LIN {X 0,Y 359.061,Z 1104.275,A -85,B 0,C 180,E1 17031.739,E2 17031.739} C_VEL
LIN {X 0,Y 356.222,Z 1112.102,A -85,B 0,C 180,E1 17028.323,E2 17028.323} C_VEL
LIN {X 0,Y 354.093,Z 1119.043,A -85,B 0,C 180,E1 17024.556,E2 17024.556} C_VEL
LIN {X 0,Y 352.905,Z 1123.818,A -85,B 0,C 180,E1 17021.108,E2 17021.108} C_VEL
LIN {X 0,Y 352.252,Z 1127.627,A -85,B 0,C 180,E1 17017.339,E2 17017.339} C_VEL
LIN {X 0,Y 352.019,Z 1129.695,A -85,B 0,C 180,E1 17013.746,E2 17013.746} C_VEL
LIN {X 0,Y 351.982,Z 1130.473,A -85,B 0,C 180,E1 17010.488,E2 17010.488} C_VEL
LIN {X 0,Y 352.008,Z 1129.935,A -85,B 0,C 180,E1 17006.743,E2 17006.743} C_VEL
LIN {X 0,Y 352.17,Z 1128.245,A -85,B 0,C 180,E1 17003.479,E2 17003.479} C_VEL
LIN {X 0,Y 352.699,Z 1124.946,A -85,B 0,C 180,E1 16999.712,E2 16999.712} C_VEL
LIN {X 0,Y 353.78,Z 1120.188,A -85,B 0,C 180,E1 16996.099,E2 16996.099} C_VEL
LIN {X 0,Y 355.733,Z 1113.699,A -85,B 0,C 180,E1 16992.328,E2 16992.328} C_VEL
LIN {X 0,Y 358.371,Z 1106.105,A -85,B 0,C 180,E1 16988.904,E2 16988.904} C_VEL
LIN {X 0,Y 362.142,Z 1096.54,A -85,B 0,C 180,E1 16985.36,E2 16985.36} C_VEL
LIN {X 0,Y 366.491,Z 1086.054,A -85,B 0,C 180,E1 16982.19,E2 16982.19} C_VEL
LIN {X 0,Y 372.055,Z 1073.212,A -85,B 0,C 180,E1 16978.936,E2 16978.936} C_VEL
LIN {X 0,Y 377.632,Z 1060.335,A -85,B 0,C 180,E1 16976.218,E2 16976.218} C_VEL
LIN {X 0,Y 384.31,Z 1044.71,A -85,B 0,C 180,E1 16973.43,E2 16973.43} C_VEL
LIN {X 0,Y 387.935,Z 1036.089,A -85,B 0,C 180,E1 16972.084,E2 16972.084} C_VEL
LIN {X 0,Y 389.23,Z 1030.919,A -85,B 0,C 180,E1 16971.25,E2 16971.25} C_VEL
LIN {X 0,Y 389.848,Z 1018.215,A -85,B 0,C 180,E1 16968.956,E2 16968.956} C_VEL
LIN {X 0,Y 391.267,Z 1012.649,A -85,B 0,C 180,E1 16968.193,E2 16968.193} C_VEL
LIN {X 0,Y 397.679,Z 995.626,A -85,B 0,C 180,E1 16966.355,E2 16966.355} C_VEL
LIN {X 0,Y 404.403,Z 976.385,A -85,B 0,C 180,E1 16964.595,E2 16964.595} C_VEL
LIN {X 0,Y 410.42,Z 957.139,A -85,B 0,C 180,E1 16963.142,E2 16963.142} C_VEL
LIN {X 0,Y 416.404,Z 935.648,A -85,B 0,C 180,E1 16961.79,E2 16961.79} C_VEL
LIN {X 0,Y 421.3,Z 914.994,A -85,B 0,C 180,E1 16960.743,E2 16960.743} C_VEL
LIN {X 0,Y 425.894,Z 891.963,A -85,B 0,C 180,E1 16959.811,E2 16959.811} C_VEL
LIN {X 0,Y 429.214,Z 870.775,A -85,B 0,C 180,E1 16959.159,E2 16959.159} C_VEL
LIN {X 0,Y 431.994,Z 846.358,A -85,B 0,C 180,E1 16958.605,E2 16958.605} C_VEL
LIN {X 0,Y 442.006,Z 679.643,A -85,B 0,C 180,E1 16955.914,E2 16955.914} C_VEL
LIN {X 0,Y 446.907,Z 597.821,A -85,B 0,C 180,E1 16954.587,E2 16954.587} C_VEL
LIN {X 0,Y 437.742,Z 580.906,A -85,B 0,C 180,E1 16952.156,E2 16952.156} C_VEL
LIN {X 0,Y 428.866,Z 565.701,A -85,B 0,C 180,E1 16949.545,E2 16949.545} C_VEL
LIN {X 0,Y 420.78,Z 552.841,A -85,B 0,C 180,E1 16946.878,E2 16946.878} C_VEL
LIN {X 0,Y 413.2,Z 541.412,A -85,B 0,C 180,E1 16944.026,E2 16944.026} C_VEL
LIN {X 0,Y 406.985,Z 532.513,A -85,B 0,C 180,E1 16941.322,E2 16941.322} C_VEL
LIN {X 0,Y 401.123,Z 524.227,A -85,B 0,C 180,E1 16938.306,E2 16938.306} C_VEL
LIN {X 0,Y 396.734,Z 518.263,A -85,B 0,C 180,E1 16935.57,E2 16935.57} C_VEL
LIN {X 0,Y 393.297,Z 513.694,A -85,B 0,C 180,E1 16932.928,E2 16932.928} C_VEL
LIN {X 0,Y 389.738,Z 508.601,A -85,B 0,C 180,E1 16929.153,E2 16929.153} C_VEL
LIN {X 0,Y 387.106,Z 505.134,A -85,B 0,C 180,E1 16923.258,E2 16923.258} C_VEL
LIN {X 0,Y 387.254,Z 504.707,A -85,B 0,C 180,E1 16919.852,E2 16919.852} C_VEL
LIN {X 0,Y 388.647,Z 506.124,A -85,B 0,C 180,E1 16916.312,E2 16916.312} C_VEL
LIN {X 0,Y 393.194,Z 510.647,A -85,B 0,C 180,E1 16911.076,E2 16911.076} C_VEL
LIN {X 0,Y 398.383,Z 516.743,A -85,B 0,C 180,E1 16907.24,E2 16907.24} C_VEL
LIN {X 0,Y 403.316,Z 522.752,A -85,B 0,C 180,E1 16904.396,E2 16904.396} C_VEL
LIN {X 0,Y 408.456,Z 529.319,A -85,B 0,C 180,E1 16901.887,E2 16901.887} C_VEL
LIN {X 0,Y 414.502,Z 537.176,A -85,B 0,C 180,E1 16899.342,E2 16899.342} C_VEL
LIN {X 0,Y 421.272,Z 546.488,A -85,B 0,C 180,E1 16896.833,E2 16896.833} C_VEL
LIN {X 0,Y 430.458,Z 559.864,A -85,B 0,C 180,E1 16893.847,E2 16893.847} C_VEL
LIN {X 0,Y 439.172,Z 573.641,A -85,B 0,C 180,E1 16891.326,E2 16891.326} C_VEL
LIN {X 0,Y 448.301,Z 589.215,A -85,B 0,C 180,E1 16888.931,E2 16888.931} C_VEL
LIN {X 0,Y 448.71,Z 590.437,A -85,B 0,C 180,E1 16888.814,E2 16888.814} C_VEL
LIN {X 0,Y 434.047,Z 817.562,A -85,B 0,C 180,E1 16885.027,E2 16885.027} C_VEL
LIN {X 0,Y 431.532,Z 850.715,A -85,B 0,C 180,E1 16884.419,E2 16884.419} C_VEL
LIN {X 0,Y 428.713,Z 872.916,A -85,B 0,C 180,E1 16883.861,E2 16883.861} C_VEL
LIN {X 0,Y 424.851,Z 896.32,A -85,B 0,C 180,E1 16883.093,E2 16883.093} C_VEL
LIN {X 0,Y 420.337,Z 918.145,A -85,B 0,C 180,E1 16882.163,E2 16882.163} C_VEL
LIN {X 0,Y 414.997,Z 940.571,A -85,B 0,C 180,E1 16880.99,E2 16880.99} C_VEL
LIN {X 0,Y 409.021,Z 961.94,A -85,B 0,C 180,E1 16879.607,E2 16879.607} C_VEL
LIN {X 0,Y 402.496,Z 983.175,A -85,B 0,C 180,E1 16877.969,E2 16877.969} C_VEL
LIN {X 0,Y 395.82,Z 1002.626,A -85,B 0,C 180,E1 16876.155,E2 16876.155} C_VEL
LIN {X 0,Y 389.09,Z 1021.112,A -85,B 0,C 180,E1 16874.141,E2 16874.141} C_VEL
LIN {X 0,Y 382.174,Z 1038.777,A -85,B 0,C 180,E1 16871.849,E2 16871.849} C_VEL
LIN {X 0,Y 375.67,Z 1054.927,A -85,B 0,C 180,E1 16869.405,E2 16869.405} C_VEL
LIN {X 0,Y 368.791,Z 1071.506,A -85,B 0,C 180,E1 16866.425,E2 16866.425} C_VEL
LIN {X 0,Y 362.918,Z 1085.776,A -85,B 0,C 180,E1 16863.404,E2 16863.404} C_VEL
LIN {X 0,Y 357.509,Z 1099.067,A -85,B 0,C 180,E1 16860.042,E2 16860.042} C_VEL
LIN {X 0,Y 353.277,Z 1110.136,A -85,B 0,C 180,E1 16856.745,E2 16856.745} C_VEL
LIN {X 0,Y 349.514,Z 1120.844,A -85,B 0,C 180,E1 16852.897,E2 16852.897} C_VEL
LIN {X 0,Y 347.053,Z 1128.999,A -85,B 0,C 180,E1 16849.349,E2 16849.349} C_VEL
LIN {X 0,Y 345.234,Z 1136.464,A -85,B 0,C 180,E1 16845.281,E2 16845.281} C_VEL
LIN {X 0,Y 344.401,Z 1141.286,A -85,B 0,C 180,E1 16841.896,E2 16841.896} C_VEL
LIN {X 0,Y 344.011,Z 1145.264,A -85,B 0,C 180,E1 16838.188,E2 16838.188} C_VEL
LIN {X 0,Y 343.957,Z 1147.712,A -85,B 0,C 180,E1 16834.354,E2 16834.354} C_VEL
LIN {X 0,Y 343.97,Z 1148.635,A -85,B 0,C 180,E1 16831.166,E2 16831.166} C_VEL
LIN {X 0,Y 343.967,Z 1148.513,A -85,B 0,C 180,E1 16828.001,E2 16828.001} C_VEL
LIN {X 0,Y 343.947,Z 1147.058,A -85,B 0,C 180,E1 16824.327,E2 16824.327} C_VEL
LIN {X 0,Y 344.078,Z 1144.249,A -85,B 0,C 180,E1 16820.803,E2 16820.803} C_VEL
LIN {X 0,Y 344.527,Z 1140.404,A -85,B 0,C 180,E1 16817.428,E2 16817.428} C_VEL
LIN {X 0,Y 345.74,Z 1134.166,A -85,B 0,C 180,E1 16813.363,E2 16813.363} C_VEL
LIN {X 0,Y 347.557,Z 1127.132,A -85,B 0,C 180,E1 16809.804,E2 16809.804} C_VEL
LIN {X 0,Y 350.529,Z 1117.791,A -85,B 0,C 180,E1 16805.926,E2 16805.926} C_VEL
LIN {X 0,Y 354.257,Z 1107.381,A -85,B 0,C 180,E1 16802.408,E2 16802.408} C_VEL
LIN {X 0,Y 358.961,Z 1095.438,A -85,B 0,C 180,E1 16798.981,E2 16798.981} C_VEL
LIN {X 0,Y 364.403,Z 1081.972,A -85,B 0,C 180,E1 16795.771,E2 16795.771} C_VEL
LIN {X 0,Y 370.807,Z 1066.608,A -85,B 0,C 180,E1 16792.647,E2 16792.647} C_VEL
LIN {X 0,Y 377.109,Z 1051.19,A -85,B 0,C 180,E1 16790.021,E2 16790.021} C_VEL
LIN {X 0,Y 384.057,Z 1033.978,A -85,B 0,C 180,E1 16787.498,E2 16787.498} C_VEL
LIN {X 0,Y 391.091,Z 1015.367,A -85,B 0,C 180,E1 16785.222,E2 16785.222} C_VEL
LIN {X 0,Y 398.22,Z 995.587,A -85,B 0,C 180,E1 16783.162,E2 16783.162} C_VEL
LIN {X 0,Y 404.74,Z 975.569,A -85,B 0,C 180,E1 16781.428,E2 16781.428} C_VEL
LIN {X 0,Y 411.226,Z 954.07,A -85,B 0,C 180,E1 16779.862,E2 16779.862} C_VEL
LIN {X 0,Y 416.89,Z 932.287,A -85,B 0,C 180,E1 16778.565,E2 16778.565} C_VEL
LIN {X 0,Y 422.194,Z 909.086,A -85,B 0,C 180,E1 16777.432,E2 16777.432} C_VEL
LIN {X 0,Y 426.486,Z 886.058,A -85,B 0,C 180,E1 16776.558,E2 16776.558} C_VEL
LIN {X 0,Y 430.113,Z 861.931,A -85,B 0,C 180,E1 16775.851,E2 16775.851} C_VEL
LIN {X 0,Y 432.499,Z 838.378,A -85,B 0,C 180,E1 16775.35,E2 16775.35} C_VEL
LIN {X 0,Y 447.368,Z 608.588,A -85,B 0,C 180,E1 16771.497,E2 16771.497} C_VEL
LIN {X 0,Y 448.503,Z 589.718,A -85,B 0,C 180,E1 16771.165,E2 16771.165} C_VEL
LIN {X 0,Y 439.981,Z 575.175,A -85,B 0,C 180,E1 16768.951,E2 16768.951} C_VEL
LIN {X 0,Y 431.796,Z 562.051,A -85,B 0,C 180,E1 16766.621,E2 16766.621} C_VEL
LIN {X 0,Y 423.202,Z 549.341,A -85,B 0,C 180,E1 16763.904,E2 16763.904} C_VEL
LIN {X 0,Y 415.885,Z 539.147,A -85,B 0,C 180,E1 16761.287,E2 16761.287} C_VEL
LIN {X 0,Y 409.44,Z 530.6,A -85,B 0,C 180,E1 16758.658,E2 16758.658} C_VEL
LIN {X 0,Y 405.218,Z 525.317,A -85,B 0,C 180,E1 16756.707,E2 16756.707} C_VEL
LIN {X 0,Y 401.668,Z 520.808,A -85,B 0,C 180,E1 16754.857,E2 16754.857} C_VEL
LIN {X 0,Y 397.261,Z 515.456,A -85,B 0,C 180,E1 16752.206,E2 16752.206} C_VEL
LIN {X 0,Y 392.273,Z 509.7,A -85,B 0,C 180,E1 16748.354,E2 16748.354} C_VEL
LIN {X 0,Y 387.81,Z 505.149,A -85,B 0,C 180,E1 16742.66,E2 16742.66} C_VEL
LIN {X 0,Y 386.775,Z 504.223,A -85,B 0,C 180,E1 16739.111,E2 16739.111} C_VEL
LIN {X 0,Y 386.947,Z 505.163,A -85,B 0,C 180,E1 16735.702,E2 16735.702} C_VEL
LIN {X 0,Y 390.01,Z 509.049,A -85,B 0,C 180,E1 16730.035,E2 16730.035} C_VEL
LIN {X 0,Y 394.226,Z 515.041,A -85,B 0,C 180,E1 16725.982,E2 16725.982} C_VEL
LIN {X 0,Y 397.728,Z 519.696,A -85,B 0,C 180,E1 16723.496,E2 16723.496} C_VEL
LIN {X 0,Y 402.885,Z 526.813,A -85,B 0,C 180,E1 16720.5,E2 16720.5} C_VEL
LIN {X 0,Y 408.579,Z 534.863,A -85,B 0,C 180,E1 16717.746,E2 16717.746} C_VEL
LIN {X 0,Y 414.522,Z 543.603,A -85,B 0,C 180,E1 16715.259,E2 16715.259} C_VEL
LIN {X 0,Y 421.57,Z 554.129,A -85,B 0,C 180,E1 16712.681,E2 16712.681} C_VEL
LIN {X 0,Y 429.653,Z 567.202,A -85,B 0,C 180,E1 16710.054,E2 16710.054} C_VEL
LIN {X 0,Y 438.52,Z 582.46,A -85,B 0,C 180,E1 16707.483,E2 16707.483} C_VEL
LIN {X 0,Y 446.862,Z 597.937,A -85,B 0,C 180,E1 16705.287,E2 16705.287} C_VEL
LIN {X 0,Y 432.543,Z 837.338,A -85,B 0,C 180,E1 16701.454,E2 16701.454} C_VEL
LIN {X 0,Y 430.479,Z 859.725,A -85,B 0,C 180,E1 16701.013,E2 16701.013} C_VEL
LIN {X 0,Y 426.9,Z 885.077,A -85,B 0,C 180,E1 16700.318,E2 16700.318} C_VEL
LIN {X 0,Y 423.093,Z 905.925,A -85,B 0,C 180,E1 16699.551,E2 16699.551} C_VEL
LIN {X 0,Y 417.989,Z 928.682,A -85,B 0,C 180,E1 16698.482,E2 16698.482} C_VEL
LIN {X 0,Y 412.773,Z 948.636,A -85,B 0,C 180,E1 16697.324,E2 16697.324} C_VEL
LIN {X 0,Y 406.394,Z 969.781,A -85,B 0,C 180,E1 16695.825,E2 16695.825} C_VEL
LIN {X 0,Y 400.067,Z 988.711,A -85,B 0,C 180,E1 16694.212,E2 16694.212} C_VEL
LIN {X 0,Y 393.096,Z 1007.592,A -85,B 0,C 180,E1 16692.273,E2 16692.273} C_VEL
LIN {X 0,Y 386.548,Z 1024.183,A -85,B 0,C 180,E1 16690.263,E2 16690.263} C_VEL
LIN {X 0,Y 379.552,Z 1040.768,A -85,B 0,C 180,E1 16687.866,E2 16687.866} C_VEL
LIN {X 0,Y 373.139,Z 1055.439,A -85,B 0,C 180,E1 16685.367,E2 16685.367} C_VEL
LIN {X 0,Y 366.755,Z 1069.59,A -85,B 0,C 180,E1 16682.486,E2 16682.486} C_VEL
LIN {X 0,Y 361.236,Z 1081.899,A -85,B 0,C 180,E1 16679.518,E2 16679.518} C_VEL
LIN {X 0,Y 356.1,Z 1093.44,A -85,B 0,C 180,E1 16676.158,E2 16676.158} C_VEL
LIN {X 0,Y 352,Z 1103.261,A -85,B 0,C 180,E1 16672.726,E2 16672.726} C_VEL
LIN {X 0,Y 348.749,Z 1111.638,A -85,B 0,C 180,E1 16669.078,E2 16669.078} C_VEL
LIN {X 0,Y 346.409,Z 1118.767,A -85,B 0,C 180,E1 16665.228,E2 16665.228} C_VEL
LIN {X 0,Y 344.974,Z 1124.033,A -85,B 0,C 180,E1 16661.367,E2 16661.367} C_VEL
LIN {X 0,Y 344.278,Z 1127.839,A -85,B 0,C 180,E1 16657.51,E2 16657.51} C_VEL
LIN {X 0,Y 344.026,Z 1129.906,A -85,B 0,C 180,E1 16653.833,E2 16653.833} C_VEL
LIN {X 0,Y 343.986,Z 1130.683,A -85,B 0,C 180,E1 16650.5,E2 16650.5} C_VEL
LIN {X 0,Y 344.014,Z 1130.145,A -85,B 0,C 180,E1 16646.667,E2 16646.667} C_VEL
LIN {X 0,Y 344.189,Z 1128.456,A -85,B 0,C 180,E1 16643.327,E2 16643.327} C_VEL
LIN {X 0,Y 344.762,Z 1125.16,A -85,B 0,C 180,E1 16639.472,E2 16639.472} C_VEL
LIN {X 0,Y 345.911,Z 1120.403,A -85,B 0,C 180,E1 16635.777,E2 16635.777} C_VEL
LIN {X 0,Y 347.986,Z 1113.918,A -85,B 0,C 180,E1 16631.921,E2 16631.921} C_VEL
LIN {X 0,Y 350.775,Z 1106.327,A -85,B 0,C 180,E1 16628.425,E2 16628.425} C_VEL
LIN {X 0,Y 354.763,Z 1096.7,A -85,B 0,C 180,E1 16624.788,E2 16624.788} C_VEL
LIN {X 0,Y 359.314,Z 1086.226,A -85,B 0,C 180,E1 16621.565,E2 16621.565} C_VEL
LIN {X 0,Y 365.092,Z 1073.454,A -85,B 0,C 180,E1 16618.275,E2 16618.275} C_VEL
LIN {X 0,Y 370.883,Z 1060.583,A -85,B 0,C 180,E1 16615.517,E2 16615.517} C_VEL
LIN {X 0,Y 377.812,Z 1044.976,A -85,B 0,C 180,E1 16612.695,E2 16612.695} C_VEL
LIN {X 0,Y 384.289,Z 1029.794,A -85,B 0,C 180,E1 16610.396,E2 16610.396} C_VEL
LIN {X 0,Y 391.267,Z 1012.649,A -85,B 0,C 180,E1 16608.193,E2 16608.193} C_VEL
LIN {X 0,Y 392.706,Z 1006.997,A -85,B 0,C 180,E1 16607.447,E2 16607.447} C_VEL
LIN {X 0,Y 393.841,Z 992.179,A -85,B 0,C 180,E1 16605.237,E2 16605.237} C_VEL
LIN {X 0,Y 395.183,Z 986.942,A -85,B 0,C 180,E1 16604.67,E2 16604.67} C_VEL
LIN {X 0,Y 401.436,Z 968.72,A -85,B 0,C 180,E1 16603.13,E2 16603.13} C_VEL
LIN {X 0,Y 408.259,Z 946.388,A -85,B 0,C 180,E1 16601.574,E2 16601.574} C_VEL
LIN {X 0,Y 413.677,Z 926.027,A -85,B 0,C 180,E1 16600.414,E2 16600.414} C_VEL
LIN {X 0,Y 418.633,Z 903.902,A -85,B 0,C 180,E1 16599.406,E2 16599.406} C_VEL
LIN {X 0,Y 422.618,Z 882.306,A -85,B 0,C 180,E1 16598.629,E2 16598.629} C_VEL
LIN {X 0,Y 425.943,Z 858.501,A -85,B 0,C 180,E1 16597.999,E2 16597.999} C_VEL
LIN {X 0,Y 428.115,Z 834.877,A -85,B 0,C 180,E1 16597.54,E2 16597.54} C_VEL
LIN {X 0,Y 442.467,Z 601.906,A -85,B 0,C 180,E1 16593.803,E2 16593.803} C_VEL
LIN {X 0,Y 434.281,Z 586.594,A -85,B 0,C 180,E1 16591.549,E2 16591.549} C_VEL
LIN {X 0,Y 426.093,Z 572.293,A -85,B 0,C 180,E1 16589.062,E2 16589.062} C_VEL
LIN {X 0,Y 418.175,Z 559.46,A -85,B 0,C 180,E1 16586.369,E2 16586.369} C_VEL
LIN {X 0,Y 410.619,Z 547.848,A -85,B 0,C 180,E1 16583.424,E2 16583.424} C_VEL
LIN {X 0,Y 405.012,Z 539.706,A -85,B 0,C 180,E1 16580.9,E2 16580.9} C_VEL
LIN {X 0,Y 399.558,Z 531.806,A -85,B 0,C 180,E1 16578.01,E2 16578.01} C_VEL
LIN {X 0,Y 395.256,Z 525.844,A -85,B 0,C 180,E1 16575.254,E2 16575.254} C_VEL
LIN {X 0,Y 391.997,Z 521.416,A -85,B 0,C 180,E1 16572.672,E2 16572.672} C_VEL
LIN {X 0,Y 388.661,Z 516.485,A -85,B 0,C 180,E1 16569.029,E2 16569.029} C_VEL
LIN {X 0,Y 386.113,Z 513.037,A -85,B 0,C 180,E1 16563.117,E2 16563.117} C_VEL
LIN {X 0,Y 386.31,Z 512.683,A -85,B 0,C 180,E1 16559.703,E2 16559.703} C_VEL
LIN {X 0,Y 387.663,Z 514.115,A -85,B 0,C 180,E1 16556.303,E2 16556.303} C_VEL
LIN {X 0,Y 391.966,Z 518.445,A -85,B 0,C 180,E1 16551.27,E2 16551.27} C_VEL
LIN {X 0,Y 396.954,Z 524.439,A -85,B 0,C 180,E1 16547.489,E2 16547.489} C_VEL
LIN {X 0,Y 401.673,Z 530.29,A -85,B 0,C 180,E1 16544.7,E2 16544.7} C_VEL
LIN {X 0,Y 406.721,Z 536.861,A -85,B 0,C 180,E1 16542.177,E2 16542.177} C_VEL
LIN {X 0,Y 412.667,Z 544.776,A -85,B 0,C 180,E1 16539.616,E2 16539.616} C_VEL
LIN {X 0,Y 419.077,Z 553.762,A -85,B 0,C 180,E1 16537.188,E2 16537.188} C_VEL
LIN {X 0,Y 427.821,Z 566.732,A -85,B 0,C 180,E1 16534.27,E2 16534.27} C_VEL
LIN {X 0,Y 436.18,Z 580.196,A -85,B 0,C 180,E1 16531.783,E2 16531.783} C_VEL
LIN {X 0,Y 444.153,Z 594.081,A -85,B 0,C 180,E1 16529.622,E2 16529.622} C_VEL
LIN {X 0,Y 428.924,Z 823.697,A -85,B 0,C 180,E1 16525.783,E2 16525.783} C_VEL
LIN {X 0,Y 426.432,Z 853.288,A -85,B 0,C 180,E1 16525.219,E2 16525.219} C_VEL
LIN {X 0,Y 423.499,Z 875.318,A -85,B 0,C 180,E1 16524.652,E2 16524.652} C_VEL
LIN {X 0,Y 419.11,Z 900.128,A -85,B 0,C 180,E1 16523.802,E2 16523.802} C_VEL
LIN {X 0,Y 414.814,Z 920.165,A -85,B 0,C 180,E1 16522.927,E2 16522.927} C_VEL
LIN {X 0,Y 408.772,Z 944.174,A -85,B 0,C 180,E1 16521.626,E2 16521.626} C_VEL
LIN {X 0,Y 403.199,Z 963.438,A -85,B 0,C 180,E1 16520.355,E2 16520.355} C_VEL
LIN {X 0,Y 396.266,Z 985.057,A -85,B 0,C 180,E1 16518.649,E2 16518.649} C_VEL
LIN {X 0,Y 389.677,Z 1003.651,A -85,B 0,C 180,E1 16516.888,E2 16516.888} C_VEL
LIN {X 0,Y 382.289,Z 1023.139,A -85,B 0,C 180,E1 16514.715,E2 16514.715} C_VEL
LIN {X 0,Y 375.203,Z 1040.555,A -85,B 0,C 180,E1 16512.395,E2 16512.395} C_VEL
LIN {X 0,Y 367.954,Z 1057.843,A -85,B 0,C 180,E1 16509.688,E2 16509.688} C_VEL
LIN {X 0,Y 361.467,Z 1072.824,A -85,B 0,C 180,E1 16506.889,E2 16506.889} C_VEL
LIN {X 0,Y 355.185,Z 1087.473,A -85,B 0,C 180,E1 16503.682,E2 16503.682} C_VEL
LIN {X 0,Y 349.717,Z 1100.347,A -85,B 0,C 180,E1 16500.292,E2 16500.292} C_VEL
LIN {X 0,Y 345.114,Z 1111.95,A -85,B 0,C 180,E1 16496.685,E2 16496.685} C_VEL
LIN {X 0,Y 341.623,Z 1121.453,A -85,B 0,C 180,E1 16493.092,E2 16493.092} C_VEL
LIN {X 0,Y 338.898,Z 1130.216,A -85,B 0,C 180,E1 16489.117,E2 16489.117} C_VEL
LIN {X 0,Y 337.232,Z 1136.774,A -85,B 0,C 180,E1 16485.301,E2 16485.301} C_VEL
LIN {X 0,Y 336.391,Z 1141.5,A -85,B 0,C 180,E1 16481.835,E2 16481.835} C_VEL
LIN {X 0,Y 335.991,Z 1145.436,A -85,B 0,C 180,E1 16477.868,E2 16477.868} C_VEL
LIN {X 0,Y 335.961,Z 1147.581,A -85,B 0,C 180,E1 16474.267,E2 16474.267} C_VEL
LIN {X 0,Y 335.971,Z 1148.449,A -85,B 0,C 180,E1 16471.023,E2 16471.023} C_VEL
LIN {X 0,Y 335.953,Z 1148.23,A -85,B 0,C 180,E1 16467.441,E2 16467.441} C_VEL
LIN {X 0,Y 335.972,Z 1146.373,A -85,B 0,C 180,E1 16463.506,E2 16463.506} C_VEL
LIN {X 0,Y 336.148,Z 1143.536,A -85,B 0,C 180,E1 16460.065,E2 16460.065} C_VEL
LIN {X 0,Y 336.839,Z 1138.854,A -85,B 0,C 180,E1 16456.087,E2 16456.087} C_VEL
LIN {X 0,Y 338.253,Z 1132.467,A -85,B 0,C 180,E1 16452.148,E2 16452.148} C_VEL
LIN {X 0,Y 340.676,Z 1124.324,A -85,B 0,C 180,E1 16448.115,E2 16448.115} C_VEL
LIN {X 0,Y 344.01,Z 1114.727,A -85,B 0,C 180,E1 16444.337,E2 16444.337} C_VEL
LIN {X 0,Y 348.454,Z 1103.461,A -85,B 0,C 180,E1 16440.614,E2 16440.614} C_VEL
LIN {X 0,Y 353.465,Z 1091.288,A -85,B 0,C 180,E1 16437.295,E2 16437.295} C_VEL
LIN {X 0,Y 359.585,Z 1077.194,A -85,B 0,C 180,E1 16434.016,E2 16434.016} C_VEL
LIN {X 0,Y 366.059,Z 1062.027,A -85,B 0,C 180,E1 16431.079,E2 16431.079} C_VEL
LIN {X 0,Y 373.309,Z 1045.042,A -85,B 0,C 180,E1 16428.272,E2 16428.272} C_VEL
LIN {X 0,Y 380.437,Z 1027.457,A -85,B 0,C 180,E1 16425.85,E2 16425.85} C_VEL
LIN {X 0,Y 387.94,Z 1008.17,A -85,B 0,C 180,E1 16423.592,E2 16423.592} C_VEL
LIN {X 0,Y 394.682,Z 989.272,A -85,B 0,C 180,E1 16421.747,E2 16421.747} C_VEL
LIN {X 0,Y 401.548,Z 968.592,A -85,B 0,C 180,E1 16420.03,E2 16420.03} C_VEL
LIN {X 0,Y 407.613,Z 947.896,A -85,B 0,C 180,E1 16418.62,E2 16418.62} C_VEL
LIN {X 0,Y 413.327,Z 926.077,A -85,B 0,C 180,E1 16417.374,E2 16417.374} C_VEL
LIN {X 0,Y 418.318,Z 903.333,A -85,B 0,C 180,E1 16416.339,E2 16416.339} C_VEL
LIN {X 0,Y 422.661,Z 879.915,A -85,B 0,C 180,E1 16415.494,E2 16415.494} C_VEL
LIN {X 0,Y 425.998,Z 855.787,A -85,B 0,C 180,E1 16414.852,E2 16414.852} C_VEL
LIN {X 0,Y 428.309,Z 831.084,A -85,B 0,C 180,E1 16414.356,E2 16414.356} C_VEL
LIN {X 0,Y 443.62,Z 599.589,A -85,B 0,C 180,E1 16410.482,E2 16410.482} C_VEL
LIN {X 0,Y 443.957,Z 593.754,A -85,B 0,C 180,E1 16410.373,E2 16410.373} C_VEL
LIN {X 0,Y 434.757,Z 577.99,A -85,B 0,C 180,E1 16407.869,E2 16407.869} C_VEL
LIN {X 0,Y 427.152,Z 565.836,A -85,B 0,C 180,E1 16405.587,E2 16405.587} C_VEL
LIN {X 0,Y 418.177,Z 552.483,A -85,B 0,C 180,E1 16402.567,E2 16402.567} C_VEL
LIN {X 0,Y 410.693,Z 542.113,A -85,B 0,C 180,E1 16399.669,E2 16399.669} C_VEL
LIN {X 0,Y 404.089,Z 533.48,A -85,B 0,C 180,E1 16396.681,E2 16396.681} C_VEL
LIN {X 0,Y 400.05,Z 528.361,A -85,B 0,C 180,E1 16394.548,E2 16394.548} C_VEL
LIN {X 0,Y 395.847,Z 523.157,A -85,B 0,C 180,E1 16391.954,E2 16391.954} C_VEL
LIN {X 0,Y 391.136,Z 517.574,A -85,B 0,C 180,E1 16388.231,E2 16388.231} C_VEL
LIN {X 0,Y 386.829,Z 513.107,A -85,B 0,C 180,E1 16382.667,E2 16382.667} C_VEL
LIN {X 0,Y 385.819,Z 512.156,A -85,B 0,C 180,E1 16379.258,E2 16379.258} C_VEL
LIN {X 0,Y 385.941,Z 513.05,A -85,B 0,C 180,E1 16375.84,E2 16375.84} C_VEL
LIN {X 0,Y 388.918,Z 516.959,A -85,B 0,C 180,E1 16370.156,E2 16370.156} C_VEL
LIN {X 0,Y 392.899,Z 522.741,A -85,B 0,C 180,E1 16366.234,E2 16366.234} C_VEL
LIN {X 0,Y 396.322,Z 527.441,A -85,B 0,C 180,E1 16363.737,E2 16363.737} C_VEL
LIN {X 0,Y 401.266,Z 534.375,A -85,B 0,C 180,E1 16360.796,E2 16360.796} C_VEL
LIN {X 0,Y 406.783,Z 542.37,A -85,B 0,C 180,E1 16358.061,E2 16358.061} C_VEL
LIN {X 0,Y 412.381,Z 550.762,A -85,B 0,C 180,E1 16355.657,E2 16355.657} C_VEL
LIN {X 0,Y 419.21,Z 561.197,A -85,B 0,C 180,E1 16353.09,E2 16353.09} C_VEL
LIN {X 0,Y 426.958,Z 573.958,A -85,B 0,C 180,E1 16350.502,E2 16350.502} C_VEL
LIN {X 0,Y 435.464,Z 588.887,A -85,B 0,C 180,E1 16347.967,E2 16347.967} C_VEL
LIN {X 0,Y 442.306,Z 601.969,A -85,B 0,C 180,E1 16346.092,E2 16346.092} C_VEL
LIN {X 0,Y 427.4,Z 842.164,A -85,B 0,C 180,E1 16342.225,E2 16342.225} C_VEL
LIN {X 0,Y 424.928,Z 865.952,A -85,B 0,C 180,E1 16341.725,E2 16341.725} C_VEL
LIN {X 0,Y 421.435,Z 888.354,A -85,B 0,C 180,E1 16341.066,E2 16341.066} C_VEL
LIN {X 0,Y 417.061,Z 910.907,A -85,B 0,C 180,E1 16340.199,E2 16340.199} C_VEL
LIN {X 0,Y 412.161,Z 931.437,A -85,B 0,C 180,E1 16339.192,E2 16339.192} C_VEL
LIN {X 0,Y 406.281,Z 952.907,A -85,B 0,C 180,E1 16337.904,E2 16337.904} C_VEL
LIN {X 0,Y 400.038,Z 972.572,A -85,B 0,C 180,E1 16336.457,E2 16336.457} C_VEL
LIN {X 0,Y 393.073,Z 992.503,A -85,B 0,C 180,E1 16334.697,E2 16334.697} C_VEL
LIN {X 0,Y 386.229,Z 1010.244,A -85,B 0,C 180,E1 16332.811,E2 16332.811} C_VEL
LIN {X 0,Y 378.645,Z 1028.577,A -85,B 0,C 180,E1 16330.489,E2 16330.489} C_VEL
LIN {X 0,Y 371.95,Z 1043.768,A -85,B 0,C 180,E1 16328.192,E2 16328.192} C_VEL
LIN {X 0,Y 364.345,Z 1060.361,A -85,B 0,C 180,E1 16325.192,E2 16325.192} C_VEL
LIN {X 0,Y 358.314,Z 1073.269,A -85,B 0,C 180,E1 16322.397,E2 16322.397} C_VEL
LIN {X 0,Y 352.239,Z 1086.178,A -85,B 0,C 180,E1 16319.036,E2 16319.036} C_VEL
LIN {X 0,Y 347.248,Z 1097.184,A -85,B 0,C 180,E1 16315.59,E2 16315.59} C_VEL
LIN {X 0,Y 343.112,Z 1106.689,A -85,B 0,C 180,E1 16311.902,E2 16311.902} C_VEL
LIN {X 0,Y 340.078,Z 1114.592,A -85,B 0,C 180,E1 16308.159,E2 16308.159} C_VEL
LIN {X 0,Y 337.944,Z 1120.95,A -85,B 0,C 180,E1 16304.216,E2 16304.216} C_VEL
LIN {X 0,Y 336.725,Z 1125.788,A -85,B 0,C 180,E1 16300.263,E2 16300.263} C_VEL
LIN {X 0,Y 336.181,Z 1128.812,A -85,B 0,C 180,E1 16296.49,E2 16296.49} C_VEL
LIN {X 0,Y 336.005,Z 1130.574,A -85,B 0,C 180,E1 16292.729,E2 16292.729} C_VEL
LIN {X 0,Y 335.987,Z 1130.841,A -85,B 0,C 180,E1 16288.977,E2 16288.977} C_VEL
LIN {X 0,Y 336.043,Z 1130.029,A -85,B 0,C 180,E1 16285.734,E2 16285.734} C_VEL
LIN {X 0,Y 336.361,Z 1127.731,A -85,B 0,C 180,E1 16281.797,E2 16281.797} C_VEL
LIN {X 0,Y 337.13,Z 1123.979,A -85,B 0,C 180,E1 16278.017,E2 16278.017} C_VEL
LIN {X 0,Y 338.715,Z 1118.601,A -85,B 0,C 180,E1 16274.065,E2 16274.065} C_VEL
LIN {X 0,Y 341.134,Z 1111.739,A -85,B 0,C 180,E1 16270.301,E2 16270.301} C_VEL
LIN {X 0,Y 344.771,Z 1102.878,A -85,B 0,C 180,E1 16266.408,E2 16266.408} C_VEL
LIN {X 0,Y 349.148,Z 1092.979,A -85,B 0,C 180,E1 16262.913,E2 16262.913} C_VEL
LIN {X 0,Y 354.875,Z 1080.664,A -85,B 0,C 180,E1 16259.337,E2 16259.337} C_VEL
LIN {X 0,Y 360.418,Z 1068.892,A -85,B 0,C 180,E1 16256.49,E2 16256.49} C_VEL
LIN {X 0,Y 367.498,Z 1053.723,A -85,B 0,C 180,E1 16253.426,E2 16253.426} C_VEL
LIN {X 0,Y 373.828,Z 1039.776,A -85,B 0,C 180,E1 16251.056,E2 16251.056} C_VEL
LIN {X 0,Y 381.254,Z 1022.611,A -85,B 0,C 180,E1 16248.597,E2 16248.597} C_VEL
LIN {X 0,Y 387.922,Z 1006.245,A -85,B 0,C 180,E1 16246.625,E2 16246.625} C_VEL
LIN {X 0,Y 395.183,Z 986.942,A -85,B 0,C 180,E1 16244.67,E2 16244.67} C_VEL
LIN {X 0,Y 396.663,Z 980.881,A -85,B 0,C 180,E1 16244.017,E2 16244.017} C_VEL
LIN {X 0,Y 398.034,Z 964.709,A -85,B 0,C 180,E1 16242.031,E2 16242.031} C_VEL
LIN {X 0,Y 399.243,Z 959.127,A -85,B 0,C 180,E1 16241.546,E2 16241.546} C_VEL
LIN {X 0,Y 405.336,Z 938.745,A -85,B 0,C 180,E1 16240.228,E2 16240.228} C_VEL
LIN {X 0,Y 410.622,Z 917.961,A -85,B 0,C 180,E1 16239.143,E2 16239.143} C_VEL
LIN {X 0,Y 414.997,Z 897.893,A -85,B 0,C 180,E1 16238.292,E2 16238.292} C_VEL
LIN {X 0,Y 419.115,Z 874.164,A -85,B 0,C 180,E1 16237.516,E2 16237.516} C_VEL
LIN {X 0,Y 421.964,Z 852.291,A -85,B 0,C 180,E1 16236.986,E2 16236.986} C_VEL
LIN {X 0,Y 424.436,Z 819.045,A -85,B 0,C 180,E1 16236.406,E2 16236.406} C_VEL
LIN {X 0,Y 437.983,Z 605.742,A -85,B 0,C 180,E1 16232.97,E2 16232.97} C_VEL
LIN {X 0,Y 430.056,Z 590.772,A -85,B 0,C 180,E1 16230.687,E2 16230.687} C_VEL
LIN {X 0,Y 422.778,Z 577.95,A -85,B 0,C 180,E1 16228.384,E2 16228.384} C_VEL
LIN {X 0,Y 415.17,Z 565.379,A -85,B 0,C 180,E1 16225.691,E2 16225.691} C_VEL
LIN {X 0,Y 407.325,Z 553.137,A -85,B 0,C 180,E1 16222.478,E2 16222.478} C_VEL
LIN {X 0,Y 402.648,Z 546.322,A -85,B 0,C 180,E1 16220.269,E2 16220.269} C_VEL
LIN {X 0,Y 397.857,Z 539.223,A -85,B 0,C 180,E1 16217.628,E2 16217.628} C_VEL
LIN {X 0,Y 393.791,Z 533.425,A -85,B 0,C 180,E1 16214.935,E2 16214.935} C_VEL
LIN {X 0,Y 390.703,Z 529.136,A -85,B 0,C 180,E1 16212.414,E2 16212.414} C_VEL
LIN {X 0,Y 387.472,Z 524.264,A -85,B 0,C 180,E1 16208.752,E2 16208.752} C_VEL
LIN {X 0,Y 385.122,Z 520.94,A -85,B 0,C 180,E1 16202.977,E2 16202.977} C_VEL
LIN {X 0,Y 385.368,Z 520.658,A -85,B 0,C 180,E1 16199.554,E2 16199.554} C_VEL
LIN {X 0,Y 386.763,Z 522.219,A -85,B 0,C 180,E1 16196.146,E2 16196.146} C_VEL
LIN {X 0,Y 390.743,Z 526.245,A -85,B 0,C 180,E1 16191.465,E2 16191.465} C_VEL
LIN {X 0,Y 395.533,Z 532.133,A -85,B 0,C 180,E1 16187.74,E2 16187.74} C_VEL
LIN {X 0,Y 400.165,Z 538.013,A -85,B 0,C 180,E1 16184.938,E2 16184.938} C_VEL
LIN {X 0,Y 404.996,Z 544.403,A -85,B 0,C 180,E1 16182.47,E2 16182.47} C_VEL
LIN {X 0,Y 411.003,Z 552.6,A -85,B 0,C 180,E1 16179.827,E2 16179.827} C_VEL
LIN {X 0,Y 417.334,Z 561.706,A -85,B 0,C 180,E1 16177.385,E2 16177.385} C_VEL
LIN {X 0,Y 425.399,Z 573.92,A -85,B 0,C 180,E1 16174.635,E2 16174.635} C_VEL
LIN {X 0,Y 433.322,Z 586.938,A -85,B 0,C 180,E1 16172.217,E2 16172.217} C_VEL
LIN {X 0,Y 439.646,Z 598.208,A -85,B 0,C 180,E1 16170.438,E2 16170.438} C_VEL
LIN {X 0,Y 423.969,Z 828.427,A -85,B 0,C 180,E1 16166.58,E2 16166.58} C_VEL
LIN {X 0,Y 421.594,Z 854.41,A -85,B 0,C 180,E1 16166.071,E2 16166.071} C_VEL
LIN {X 0,Y 418.438,Z 877.262,A -85,B 0,C 180,E1 16165.476,E2 16165.476} C_VEL
LIN {X 0,Y 414.077,Z 900.9,A -85,B 0,C 180,E1 16164.651,E2 16164.651} C_VEL
LIN {X 0,Y 409.667,Z 920.895,A -85,B 0,C 180,E1 16163.772,E2 16163.772} C_VEL
LIN {X 0,Y 403.471,Z 944.739,A -85,B 0,C 180,E1 16162.47,E2 16162.47} C_VEL
LIN {X 0,Y 397.755,Z 963.938,A -85,B 0,C 180,E1 16161.196,E2 16161.196} C_VEL
LIN {X 0,Y 390.318,Z 986.314,A -85,B 0,C 180,E1 16159.407,E2 16159.407} C_VEL
LIN {X 0,Y 383.852,Z 1003.998,A -85,B 0,C 180,E1 16157.714,E2 16157.714} C_VEL
LIN {X 0,Y 375.999,Z 1023.973,A -85,B 0,C 180,E1 16155.454,E2 16155.454} C_VEL
LIN {X 0,Y 368.968,Z 1040.691,A -85,B 0,C 180,E1 16153.199,E2 16153.199} C_VEL
LIN {X 0,Y 361.502,Z 1057.837,A -85,B 0,C 180,E1 16150.48,E2 16150.48} C_VEL
LIN {X 0,Y 354.675,Z 1072.984,A -85,B 0,C 180,E1 16147.609,E2 16147.609} C_VEL
LIN {X 0,Y 348.002,Z 1087.882,A -85,B 0,C 180,E1 16144.274,E2 16144.274} C_VEL
LIN {X 0,Y 342.468,Z 1100.357,A -85,B 0,C 180,E1 16140.922,E2 16140.922} C_VEL
LIN {X 0,Y 337.528,Z 1112.194,A -85,B 0,C 180,E1 16137.143,E2 16137.143} C_VEL
LIN {X 0,Y 333.886,Z 1121.645,A -85,B 0,C 180,E1 16133.472,E2 16133.472} C_VEL
LIN {X 0,Y 331.033,Z 1130.311,A -85,B 0,C 180,E1 16129.406,E2 16129.406} C_VEL
LIN {X 0,Y 329.288,Z 1136.82,A -85,B 0,C 180,E1 16125.499,E2 16125.499} C_VEL
LIN {X 0,Y 328.379,Z 1141.714,A -85,B 0,C 180,E1 16121.772,E2 16121.772} C_VEL
LIN {X 0,Y 327.983,Z 1145.462,A -85,B 0,C 180,E1 16117.709,E2 16117.709} C_VEL
LIN {X 0,Y 327.959,Z 1147.371,A -85,B 0,C 180,E1 16114.371,E2 16114.371} C_VEL
LIN {X 0,Y 327.973,Z 1148.24,A -85,B 0,C 180,E1 16111.048,E2 16111.048} C_VEL
LIN {X 0,Y 327.954,Z 1148.021,A -85,B 0,C 180,E1 16107.379,E2 16107.379} C_VEL
LIN {X 0,Y 327.974,Z 1146.279,A -85,B 0,C 180,E1 16103.523,E2 16103.523} C_VEL
LIN {X 0,Y 328.154,Z 1143.488,A -85,B 0,C 180,E1 16099.998,E2 16099.998} C_VEL
LIN {X 0,Y 328.877,Z 1138.891,A -85,B 0,C 180,E1 16095.923,E2 16095.923} C_VEL
LIN {X 0,Y 330.381,Z 1132.468,A -85,B 0,C 180,E1 16091.837,E2 16091.837} C_VEL
LIN {X 0,Y 332.761,Z 1124.859,A -85,B 0,C 180,E1 16087.938,E2 16087.938} C_VEL
LIN {X 0,Y 336.194,Z 1115.439,A -85,B 0,C 180,E1 16084.075,E2 16084.075} C_VEL
LIN {X 0,Y 340.3,Z 1105.376,A -85,B 0,C 180,E1 16080.614,E2 16080.614} C_VEL
LIN {X 0,Y 345.934,Z 1092.342,A -85,B 0,C 180,E1 16076.887,E2 16076.887} C_VEL
LIN {X 0,Y 351.522,Z 1079.882,A -85,B 0,C 180,E1 16073.885,E2 16073.885} C_VEL
LIN {X 0,Y 358.885,Z 1063.484,A -85,B 0,C 180,E1 16070.563,E2 16070.563} C_VEL
LIN {X 0,Y 365.479,Z 1048.581,A -85,B 0,C 180,E1 16068.017,E2 16068.017} C_VEL
LIN {X 0,Y 373.625,Z 1029.429,A -85,B 0,C 180,E1 16065.264,E2 16065.264} C_VEL
LIN {X 0,Y 380.557,Z 1012.26,A -85,B 0,C 180,E1 16063.187,E2 16063.187} C_VEL
LIN {X 0,Y 388.475,Z 991.143,A -85,B 0,C 180,E1 16061.049,E2 16061.049} C_VEL
LIN {X 0,Y 394.933,Z 972.331,A -85,B 0,C 180,E1 16059.448,E2 16059.448} C_VEL
LIN {X 0,Y 401.897,Z 949.81,A -85,B 0,C 180,E1 16057.862,E2 16057.862} C_VEL
LIN {X 0,Y 407.235,Z 930.121,A -85,B 0,C 180,E1 16056.711,E2 16056.711} C_VEL
LIN {X 0,Y 412.947,Z 905.644,A -85,B 0,C 180,E1 16055.553,E2 16055.553} C_VEL
LIN {X 0,Y 417.144,Z 883.875,A -85,B 0,C 180,E1 16054.747,E2 16054.747} C_VEL
LIN {X 0,Y 421.033,Z 857.852,A -85,B 0,C 180,E1 16054.022,E2 16054.022} C_VEL
LIN {X 0,Y 423.324,Z 835.091,A -85,B 0,C 180,E1 16053.553,E2 16053.553} C_VEL
LIN {X 0,Y 439.13,Z 603.343,A -85,B 0,C 180,E1 16049.659,E2 16049.659} C_VEL
LIN {X 0,Y 439.444,Z 597.744,A -85,B 0,C 180,E1 16049.55,E2 16049.55} C_VEL
LIN {X 0,Y 430.083,Z 581.622,A -85,B 0,C 180,E1 16046.884,E2 16046.884} C_VEL
LIN {X 0,Y 422.535,Z 569.652,A -85,B 0,C 180,E1 16044.501,E2 16044.501} C_VEL
LIN {X 0,Y 415.393,Z 558.919,A -85,B 0,C 180,E1 16041.981,E2 16041.981} C_VEL
LIN {X 0,Y 408.661,Z 549.362,A -85,B 0,C 180,E1 16039.288,E2 16039.288} C_VEL
LIN {X 0,Y 402.267,Z 540.857,A -85,B 0,C 180,E1 16036.313,E2 16036.313} C_VEL
LIN {X 0,Y 398.443,Z 535.912,A -85,B 0,C 180,E1 16034.237,E2 16034.237} C_VEL
LIN {X 0,Y 394.441,Z 530.857,A -85,B 0,C 180,E1 16031.701,E2 16031.701} C_VEL
LIN {X 0,Y 390,Z 525.448,A -85,B 0,C 180,E1 16028.106,E2 16028.106} C_VEL
LIN {X 0,Y 385.782,Z 520.994,A -85,B 0,C 180,E1 16022.525,E2 16022.525} C_VEL
LIN {X 0,Y 384.825,Z 520.105,A -85,B 0,C 180,E1 16019.107,E2 16019.107} C_VEL
LIN {X 0,Y 384.995,Z 521.108,A -85,B 0,C 180,E1 16015.681,E2 16015.681} C_VEL
LIN {X 0,Y 387.827,Z 524.868,A -85,B 0,C 180,E1 16010.278,E2 16010.278} C_VEL
LIN {X 0,Y 391.664,Z 530.58,A -85,B 0,C 180,E1 16006.416,E2 16006.416} C_VEL
LIN {X 0,Y 394.923,Z 535.181,A -85,B 0,C 180,E1 16003.98,E2 16003.98} C_VEL
LIN {X 0,Y 399.658,Z 541.935,A -85,B 0,C 180,E1 16001.095,E2 16001.095} C_VEL
LIN {X 0,Y 404.926,Z 549.757,A -85,B 0,C 180,E1 15998.412,E2 15998.412} C_VEL
LIN {X 0,Y 410.27,Z 557.935,A -85,B 0,C 180,E1 15996.055,E2 15996.055} C_VEL
LIN {X 0,Y 416.869,Z 568.26,A -85,B 0,C 180,E1 15993.504,E2 15993.504} C_VEL
LIN {X 0,Y 424.224,Z 580.591,A -85,B 0,C 180,E1 15990.98,E2 15990.98} C_VEL
LIN {X 0,Y 432.439,Z 595.311,A -85,B 0,C 180,E1 15988.457,E2 15988.457} C_VEL
LIN {X 0,Y 437.841,Z 605.929,A -85,B 0,C 180,E1 15986.918,E2 15986.918} C_VEL
LIN {X 0,Y 422.623,Z 843.405,A -85,B 0,C 180,E1 15983.08,E2 15983.08} C_VEL
LIN {X 0,Y 419.912,Z 867.81,A -85,B 0,C 180,E1 15982.552,E2 15982.552} C_VEL
LIN {X 0,Y 416.459,Z 889.226,A -85,B 0,C 180,E1 15981.915,E2 15981.915} C_VEL
LIN {X 0,Y 411.727,Z 912.626,A -85,B 0,C 180,E1 15980.999,E2 15980.999} C_VEL
LIN {X 0,Y 406.588,Z 933.462,A -85,B 0,C 180,E1 15979.962,E2 15979.962} C_VEL
LIN {X 0,Y 400.098,Z 955.994,A -85,B 0,C 180,E1 15978.568,E2 15978.568} C_VEL
LIN {X 0,Y 394.003,Z 974.556,A -85,B 0,C 180,E1 15977.174,E2 15977.174} C_VEL
LIN {X 0,Y 386.607,Z 994.811,A -85,B 0,C 180,E1 15975.336,E2 15975.336} C_VEL
LIN {X 0,Y 379.614,Z 1012.357,A -85,B 0,C 180,E1 15973.43,E2 15973.43} C_VEL
LIN {X 0,Y 371.89,Z 1030.237,A -85,B 0,C 180,E1 15971.101,E2 15971.101} C_VEL
LIN {X 0,Y 364.77,Z 1045.859,A -85,B 0,C 180,E1 15968.681,E2 15968.681} C_VEL
LIN {X 0,Y 357.35,Z 1061.367,A -85,B 0,C 180,E1 15965.789,E2 15965.789} C_VEL
LIN {X 0,Y 350.751,Z 1075.019,A -85,B 0,C 180,E1 15962.758,E2 15962.758} C_VEL
LIN {X 0,Y 344.584,Z 1087.523,A -85,B 0,C 180,E1 15959.367,E2 15959.367} C_VEL
LIN {X 0,Y 339.46,Z 1098.356,A -85,B 0,C 180,E1 15955.845,E2 15955.845} C_VEL
LIN {X 0,Y 335.388,Z 1107.306,A -85,B 0,C 180,E1 15952.249,E2 15952.249} C_VEL
LIN {X 0,Y 332.112,Z 1115.402,A -85,B 0,C 180,E1 15948.247,E2 15948.247} C_VEL
LIN {X 0,Y 330.088,Z 1121.166,A -85,B 0,C 180,E1 15944.562,E2 15944.562} C_VEL
LIN {X 0,Y 328.787,Z 1126,A -85,B 0,C 180,E1 15940.514,E2 15940.514} C_VEL
LIN {X 0,Y 328.201,Z 1129.024,A -85,B 0,C 180,E1 15936.648,E2 15936.648} C_VEL
LIN {X 0,Y 328.009,Z 1130.784,A -85,B 0,C 180,E1 15932.796,E2 15932.796} C_VEL
LIN {X 0,Y 327.99,Z 1131.051,A -85,B 0,C 180,E1 15928.952,E2 15928.952} C_VEL
LIN {X 0,Y 328.05,Z 1130.239,A -85,B 0,C 180,E1 15925.63,E2 15925.63} C_VEL
LIN {X 0,Y 328.391,Z 1127.943,A -85,B 0,C 180,E1 15921.596,E2 15921.596} C_VEL
LIN {X 0,Y 329.222,Z 1124.192,A -85,B 0,C 180,E1 15917.725,E2 15917.725} C_VEL
LIN {X 0,Y 330.909,Z 1118.818,A -85,B 0,C 180,E1 15913.679,E2 15913.679} C_VEL
LIN {X 0,Y 333.506,Z 1111.875,A -85,B 0,C 180,E1 15909.787,E2 15909.787} C_VEL
LIN {X 0,Y 337.307,Z 1103.102,A -85,B 0,C 180,E1 15905.853,E2 15905.853} C_VEL
LIN {X 0,Y 341.652,Z 1093.708,A -85,B 0,C 180,E1 15902.457,E2 15902.457} C_VEL
LIN {X 0,Y 347.581,Z 1081.52,A -85,B 0,C 180,E1 15898.814,E2 15898.814} C_VEL
LIN {X 0,Y 353.304,Z 1069.819,A -85,B 0,C 180,E1 15895.919,E2 15895.919} C_VEL
LIN {X 0,Y 360.607,Z 1054.808,A -85,B 0,C 180,E1 15892.809,E2 15892.809} C_VEL
LIN {X 0,Y 367.117,Z 1040.949,A -85,B 0,C 180,E1 15890.407,E2 15890.407} C_VEL
LIN {X 0,Y 375.138,Z 1023.083,A -85,B 0,C 180,E1 15887.803,E2 15887.803} C_VEL
LIN {X 0,Y 381.94,Z 1006.904,A -85,B 0,C 180,E1 15885.833,E2 15885.833} C_VEL
LIN {X 0,Y 389.789,Z 986.658,A -85,B 0,C 180,E1 15883.771,E2 15883.771} C_VEL
LIN {X 0,Y 396.264,Z 968.283,A -85,B 0,C 180,E1 15882.218,E2 15882.218} C_VEL
LIN {X 0,Y 399.243,Z 959.127,A -85,B 0,C 180,E1 15881.546,E2 15881.546} C_VEL
LIN {X 0,Y 400.771,Z 952.562,A -85,B 0,C 180,E1 15880.988,E2 15880.988} C_VEL
LIN {X 0,Y 401.708,Z 936.272,A -85,B 0,C 180,E1 15879.306,E2 15879.306} C_VEL
LIN {X 0,Y 402.832,Z 929.441,A -85,B 0,C 180,E1 15878.813,E2 15878.813} C_VEL
LIN {X 0,Y 408.386,Z 906.653,A -85,B 0,C 180,E1 15877.736,E2 15877.736} C_VEL
LIN {X 0,Y 412.618,Z 885.133,A -85,B 0,C 180,E1 15876.944,E2 15876.944} C_VEL
LIN {X 0,Y 416.465,Z 859.821,A -85,B 0,C 180,E1 15876.254,E2 15876.254} C_VEL
LIN {X 0,Y 418.686,Z 837.544,A -85,B 0,C 180,E1 15875.813,E2 15875.813} C_VEL
LIN {X 0,Y 433.644,Z 609.609,A -85,B 0,C 180,E1 15872.131,E2 15872.131} C_VEL
LIN {X 0,Y 425.627,Z 594.41,A -85,B 0,C 180,E1 15869.715,E2 15869.715} C_VEL
LIN {X 0,Y 417.708,Z 580.384,A -85,B 0,C 180,E1 15867.053,E2 15867.053} C_VEL
LIN {X 0,Y 410.328,Z 568.246,A -85,B 0,C 180,E1 15864.243,E2 15864.243} C_VEL
LIN {X 0,Y 404.258,Z 558.862,A -85,B 0,C 180,E1 15861.587,E2 15861.587} C_VEL
LIN {X 0,Y 400.865,Z 553.695,A -85,B 0,C 180,E1 15859.906,E2 15859.906} C_VEL
LIN {X 0,Y 396.305,Z 546.785,A -85,B 0,C 180,E1 15857.321,E2 15857.321} C_VEL
LIN {X 0,Y 392.338,Z 541.006,A -85,B 0,C 180,E1 15854.614,E2 15854.614} C_VEL
LIN {X 0,Y 389.418,Z 536.854,A -85,B 0,C 180,E1 15852.155,E2 15852.155} C_VEL
LIN {X 0,Y 386.404,Z 532.152,A -85,B 0,C 180,E1 15848.632,E2 15848.632} C_VEL
LIN {X 0,Y 384.133,Z 528.843,A -85,B 0,C 180,E1 15842.835,E2 15842.835} C_VEL
LIN {X 0,Y 384.429,Z 528.633,A -85,B 0,C 180,E1 15839.404,E2 15839.404} C_VEL
LIN {X 0,Y 385.781,Z 530.206,A -85,B 0,C 180,E1 15836.136,E2 15836.136} C_VEL
LIN {X 0,Y 389.597,Z 534.174,A -85,B 0,C 180,E1 15831.588,E2 15831.588} C_VEL
LIN {X 0,Y 394.221,Z 539.984,A -85,B 0,C 180,E1 15827.922,E2 15827.922} C_VEL
LIN {X 0,Y 398.543,Z 545.549,A -85,B 0,C 180,E1 15825.247,E2 15825.247} C_VEL
LIN {X 0,Y 403.564,Z 552.321,A -85,B 0,C 180,E1 15822.629,E2 15822.629} C_VEL
LIN {X 0,Y 409.827,Z 561.071,A -85,B 0,C 180,E1 15819.841,E2 15819.841} C_VEL
LIN {X 0,Y 417.013,Z 571.699,A -85,B 0,C 180,E1 15817.068,E2 15817.068} C_VEL
LIN {X 0,Y 425.706,Z 585.448,A -85,B 0,C 180,E1 15814.133,E2 15814.133} C_VEL
LIN {X 0,Y 435.059,Z 601.728,A -85,B 0,C 180,E1 15811.33,E2 15811.33} C_VEL
LIN {X 0,Y 435.199,Z 602.779,A -85,B 0,C 180,E1 15811.264,E2 15811.264} C_VEL
LIN {X 0,Y 418.997,Z 834.051,A -85,B 0,C 180,E1 15807.378,E2 15807.378} C_VEL
LIN {X 0,Y 416.651,Z 857.154,A -85,B 0,C 180,E1 15806.905,E2 15806.905} C_VEL
LIN {X 0,Y 412.942,Z 881.955,A -85,B 0,C 180,E1 15806.23,E2 15806.23} C_VEL
LIN {X 0,Y 408.597,Z 904.189,A -85,B 0,C 180,E1 15805.421,E2 15805.421} C_VEL
LIN {X 0,Y 403.149,Z 927.459,A -85,B 0,C 180,E1 15804.349,E2 15804.349} C_VEL
LIN {X 0,Y 397.369,Z 948.347,A -85,B 0,C 180,E1 15803.147,E2 15803.147} C_VEL
LIN {X 0,Y 390.393,Z 970.598,A -85,B 0,C 180,E1 15801.605,E2 15801.605} C_VEL
LIN {X 0,Y 383.709,Z 989.563,A -85,B 0,C 180,E1 15800.007,E2 15800.007} C_VEL
LIN {X 0,Y 376.299,Z 1009.066,A -85,B 0,C 180,E1 15798.074,E2 15798.074} C_VEL
LIN {X 0,Y 368.555,Z 1027.623,A -85,B 0,C 180,E1 15795.856,E2 15795.856} C_VEL
LIN {X 0,Y 360.716,Z 1045.607,A -85,B 0,C 180,E1 15793.324,E2 15793.324} C_VEL
LIN {X 0,Y 353.324,Z 1061.629,A -85,B 0,C 180,E1 15790.609,E2 15790.609} C_VEL
LIN {X 0,Y 346.194,Z 1077.023,A -85,B 0,C 180,E1 15787.548,E2 15787.548} C_VEL
LIN {X 0,Y 339.617,Z 1090.889,A -85,B 0,C 180,E1 15784.218,E2 15784.218} C_VEL
LIN {X 0,Y 333.843,Z 1103.624,A -85,B 0,C 180,E1 15780.608,E2 15780.608} C_VEL
LIN {X 0,Y 329.151,Z 1114.326,A -85,B 0,C 180,E1 15776.913,E2 15776.913} C_VEL
LIN {X 0,Y 325.409,Z 1123.924,A -85,B 0,C 180,E1 15772.969,E2 15772.969} C_VEL
LIN {X 0,Y 322.676,Z 1131.974,A -85,B 0,C 180,E1 15768.8,E2 15768.8} C_VEL
LIN {X 0,Y 321.067,Z 1138.185,A -85,B 0,C 180,E1 15764.796,E2 15764.796} C_VEL
LIN {X 0,Y 320.217,Z 1142.961,A -85,B 0,C 180,E1 15760.616,E2 15760.616} C_VEL
LIN {X 0,Y 319.989,Z 1145.845,A -85,B 0,C 180,E1 15757,E2 15757} C_VEL
LIN {X 0,Y 319.955,Z 1147.657,A -85,B 0,C 180,E1 15753.225,E2 15753.225} C_VEL
LIN {X 0,Y 319.971,Z 1148.074,A -85,B 0,C 180,E1 15749.284,E2 15749.284} C_VEL
LIN {X 0,Y 319.963,Z 1147.294,A -85,B 0,C 180,E1 15745.878,E2 15745.878} C_VEL
LIN {X 0,Y 319.98,Z 1145.473,A -85,B 0,C 180,E1 15742.458,E2 15742.458} C_VEL
LIN {X 0,Y 320.34,Z 1142.104,A -85,B 0,C 180,E1 15738.477,E2 15738.477} C_VEL
LIN {X 0,Y 321.345,Z 1136.834,A -85,B 0,C 180,E1 15734.294,E2 15734.294} C_VEL
LIN {X 0,Y 323.069,Z 1130.678,A -85,B 0,C 180,E1 15730.472,E2 15730.472} C_VEL
LIN {X 0,Y 326.157,Z 1121.781,A -85,B 0,C 180,E1 15726.13,E2 15726.13} C_VEL
LIN {X 0,Y 329.753,Z 1112.849,A -85,B 0,C 180,E1 15722.555,E2 15722.555} C_VEL
LIN {X 0,Y 335.1,Z 1100.627,A -85,B 0,C 180,E1 15718.522,E2 15718.522} C_VEL
LIN {X 0,Y 340.532,Z 1088.847,A -85,B 0,C 180,E1 15715.275,E2 15715.275} C_VEL
LIN {X 0,Y 347.768,Z 1073.376,A -85,B 0,C 180,E1 15711.714,E2 15711.714} C_VEL
LIN {X 0,Y 354.525,Z 1058.909,A -85,B 0,C 180,E1 15708.917,E2 15708.917} C_VEL
LIN {X 0,Y 362.581,Z 1041.128,A -85,B 0,C 180,E1 15706.035,E2 15706.035} C_VEL
LIN {X 0,Y 369.752,Z 1024.618,A -85,B 0,C 180,E1 15703.778,E2 15703.778} C_VEL
LIN {X 0,Y 377.824,Z 1004.787,A -85,B 0,C 180,E1 15701.501,E2 15701.501} C_VEL
LIN {X 0,Y 384.623,Z 986.739,A -85,B 0,C 180,E1 15699.756,E2 15699.756} C_VEL
LIN {X 0,Y 392.086,Z 965.028,A -85,B 0,C 180,E1 15698,E2 15698} C_VEL
LIN {X 0,Y 397.935,Z 945.962,A -85,B 0,C 180,E1 15696.721,E2 15696.721} C_VEL
LIN {X 0,Y 403.97,Z 923.746,A -85,B 0,C 180,E1 15695.479,E2 15695.479} C_VEL
LIN {X 0,Y 408.92,Z 902.014,A -85,B 0,C 180,E1 15694.509,E2 15694.509} C_VEL
LIN {X 0,Y 413.461,Z 878.273,A -85,B 0,C 180,E1 15693.67,E2 15693.67} C_VEL
LIN {X 0,Y 416.777,Z 854.903,A -85,B 0,C 180,E1 15693.058,E2 15693.058} C_VEL
LIN {X 0,Y 419.2,Z 829.39,A -85,B 0,C 180,E1 15692.554,E2 15692.554} C_VEL
LIN {X 0,Y 435.087,Z 602.117,A -85,B 0,C 180,E1 15688.738,E2 15688.738} C_VEL
LIN {X 0,Y 427.406,Z 588.495,A -85,B 0,C 180,E1 15686.466,E2 15686.466} C_VEL
LIN {X 0,Y 420.175,Z 576.811,A -85,B 0,C 180,E1 15684.124,E2 15684.124} C_VEL
LIN {X 0,Y 413.165,Z 566.044,A -85,B 0,C 180,E1 15681.583,E2 15681.583} C_VEL
LIN {X 0,Y 406.497,Z 556.411,A -85,B 0,C 180,E1 15678.835,E2 15678.835} C_VEL
LIN {X 0,Y 400.33,Z 548.072,A -85,B 0,C 180,E1 15675.872,E2 15675.872} C_VEL
LIN {X 0,Y 396.97,Z 543.591,A -85,B 0,C 180,E1 15673.993,E2 15673.993} C_VEL
LIN {X 0,Y 393.042,Z 538.556,A -85,B 0,C 180,E1 15671.445,E2 15671.445} C_VEL
LIN {X 0,Y 388.712,Z 533.199,A -85,B 0,C 180,E1 15667.836,E2 15667.836} C_VEL
LIN {X 0,Y 384.739,Z 528.881,A -85,B 0,C 180,E1 15662.383,E2 15662.383} C_VEL
LIN {X 0,Y 383.834,Z 528.053,A -85,B 0,C 180,E1 15658.955,E2 15658.955} C_VEL
LIN {X 0,Y 384.053,Z 529.163,A -85,B 0,C 180,E1 15655.52,E2 15655.52} C_VEL
LIN {X 0,Y 386.739,Z 532.776,A -85,B 0,C 180,E1 15650.4,E2 15650.4} C_VEL
LIN {X 0,Y 390.347,Z 538.278,A -85,B 0,C 180,E1 15646.671,E2 15646.671} C_VEL
LIN {X 0,Y 393.433,Z 542.738,A -85,B 0,C 180,E1 15644.296,E2 15644.296} C_VEL
LIN {X 0,Y 398.184,Z 549.679,A -85,B 0,C 180,E1 15641.327,E2 15641.327} C_VEL
LIN {X 0,Y 403.156,Z 557.258,A -85,B 0,C 180,E1 15638.732,E2 15638.732} C_VEL
LIN {X 0,Y 408.161,Z 565.079,A -85,B 0,C 180,E1 15636.465,E2 15636.465} C_VEL
LIN {X 0,Y 414.553,Z 575.32,A -85,B 0,C 180,E1 15633.923,E2 15633.923} C_VEL
LIN {X 0,Y 421.56,Z 587.298,A -85,B 0,C 180,E1 15631.449,E2 15631.449} C_VEL
LIN {X 0,Y 429.419,Z 601.693,A -85,B 0,C 180,E1 15628.96,E2 15628.96} C_VEL
LIN {X 0,Y 433.473,Z 609.785,A -85,B 0,C 180,E1 15627.763,E2 15627.763} C_VEL
LIN {X 0,Y 417.999,Z 843.958,A -85,B 0,C 180,E1 15623.967,E2 15623.967} C_VEL
LIN {X 0,Y 415.064,Z 869.14,A -85,B 0,C 180,E1 15623.413,E2 15623.413} C_VEL
LIN {X 0,Y 411.546,Z 890.282,A -85,B 0,C 180,E1 15622.778,E2 15622.778} C_VEL
LIN {X 0,Y 406.749,Z 913.197,A -85,B 0,C 180,E1 15621.873,E2 15621.873} C_VEL
LIN {X 0,Y 401.694,Z 933.19,A -85,B 0,C 180,E1 15620.878,E2 15620.878} C_VEL
LIN {X 0,Y 395.124,Z 955.513,A -85,B 0,C 180,E1 15619.503,E2 15619.503} C_VEL
LIN {X 0,Y 388.859,Z 974.13,A -85,B 0,C 180,E1 15618.108,E2 15618.108} C_VEL
LIN {X 0,Y 380.98,Z 995.138,A -85,B 0,C 180,E1 15616.199,E2 15616.199} C_VEL
LIN {X 0,Y 373.784,Z 1012.665,A -85,B 0,C 180,E1 15614.282,E2 15614.282} C_VEL
LIN {X 0,Y 365.821,Z 1030.517,A -85,B 0,C 180,E1 15611.935,E2 15611.935} C_VEL
LIN {X 0,Y 358.468,Z 1046.13,A -85,B 0,C 180,E1 15609.492,E2 15609.492} C_VEL
LIN {X 0,Y 351.158,Z 1060.862,A -85,B 0,C 180,E1 15606.724,E2 15606.724} C_VEL
LIN {X 0,Y 344.648,Z 1073.76,A -85,B 0,C 180,E1 15603.851,E2 15603.851} C_VEL
LIN {X 0,Y 338.063,Z 1086.635,A -85,B 0,C 180,E1 15600.383,E2 15600.383} C_VEL
LIN {X 0,Y 332.594,Z 1097.647,A -85,B 0,C 180,E1 15596.805,E2 15596.805} C_VEL
LIN {X 0,Y 328.031,Z 1107.136,A -85,B 0,C 180,E1 15592.965,E2 15592.965} C_VEL
LIN {X 0,Y 324.521,Z 1115.326,A -85,B 0,C 180,E1 15588.876,E2 15588.876} C_VEL
LIN {X 0,Y 322.243,Z 1121.382,A -85,B 0,C 180,E1 15584.924,E2 15584.924} C_VEL
LIN {X 0,Y 320.855,Z 1126.213,A -85,B 0,C 180,E1 15580.777,E2 15580.777} C_VEL
LIN {X 0,Y 320.218,Z 1129.245,A -85,B 0,C 180,E1 15576.798,E2 15576.798} C_VEL
LIN {X 0,Y 320.013,Z 1130.995,A -85,B 0,C 180,E1 15572.866,E2 15572.866} C_VEL
LIN {X 0,Y 319.993,Z 1131.261,A -85,B 0,C 180,E1 15568.926,E2 15568.926} C_VEL
LIN {X 0,Y 320.058,Z 1130.45,A -85,B 0,C 180,E1 15565.52,E2 15565.52} C_VEL
LIN {X 0,Y 320.423,Z 1128.155,A -85,B 0,C 180,E1 15561.385,E2 15561.385} C_VEL
LIN {X 0,Y 321.321,Z 1124.406,A -85,B 0,C 180,E1 15557.419,E2 15557.419} C_VEL
LIN {X 0,Y 323.117,Z 1119.035,A -85,B 0,C 180,E1 15553.274,E2 15553.274} C_VEL
LIN {X 0,Y 325.832,Z 1112.176,A -85,B 0,C 180,E1 15549.335,E2 15549.335} C_VEL
LIN {X 0,Y 329.875,Z 1103.326,A -85,B 0,C 180,E1 15545.273,E2 15545.273} C_VEL
LIN {X 0,Y 334.43,Z 1093.935,A -85,B 0,C 180,E1 15541.81,E2 15541.81} C_VEL
LIN {X 0,Y 340.621,Z 1081.756,A -85,B 0,C 180,E1 15538.103,E2 15538.103} C_VEL
LIN {X 0,Y 346.94,Z 1069.371,A -85,B 0,C 180,E1 15535.004,E2 15535.004} C_VEL
LIN {X 0,Y 354.558,Z 1054.233,A -85,B 0,C 180,E1 15531.859,E2 15531.859} C_VEL
LIN {X 0,Y 361.332,Z 1040.3,A -85,B 0,C 180,E1 15529.435,E2 15529.435} C_VEL
LIN {X 0,Y 369.656,Z 1022.275,A -85,B 0,C 180,E1 15526.816,E2 15526.816} C_VEL
LIN {X 0,Y 376.885,Z 1005.574,A -85,B 0,C 180,E1 15524.79,E2 15524.79} C_VEL
LIN {X 0,Y 384.532,Z 986.271,A -85,B 0,C 180,E1 15522.838,E2 15522.838} C_VEL
LIN {X 0,Y 391.478,Z 967.061,A -85,B 0,C 180,E1 15521.222,E2 15521.222} C_VEL
LIN {X 0,Y 398.131,Z 946.169,A -85,B 0,C 180,E1 15519.78,E2 15519.78} C_VEL
LIN {X 0,Y 402.832,Z 929.441,A -85,B 0,C 180,E1 15518.813,E2 15518.813} C_VEL
LIN {X 0,Y 404.098,Z 922.514,A -85,B 0,C 180,E1 15518.345,E2 15518.345} C_VEL
LIN {X 0,Y 404.615,Z 905.262,A -85,B 0,C 180,E1 15516.884,E2 15516.884} C_VEL
LIN {X 0,Y 405.533,Z 898.12,A -85,B 0,C 180,E1 15516.481,E2 15516.481} C_VEL
LIN {X 0,Y 409.881,Z 874.28,A -85,B 0,C 180,E1 15515.704,E2 15515.704} C_VEL
LIN {X 0,Y 412.859,Z 852.461,A -85,B 0,C 180,E1 15515.176,E2 15515.176} C_VEL
LIN {X 0,Y 415.467,Z 819.512,A -85,B 0,C 180,E1 15514.598,E2 15514.598} C_VEL
LIN {X 0,Y 429.351,Z 613.526,A -85,B 0,C 180,E1 15511.265,E2 15511.265} C_VEL
LIN {X 0,Y 421.32,Z 598.124,A -85,B 0,C 180,E1 15508.723,E2 15508.723} C_VEL
LIN {X 0,Y 414.29,Z 585.732,A -85,B 0,C 180,E1 15506.249,E2 15506.249} C_VEL
LIN {X 0,Y 408.132,Z 575.285,A -85,B 0,C 180,E1 15503.805,E2 15503.805} C_VEL
LIN {X 0,Y 402.345,Z 566.13,A -85,B 0,C 180,E1 15501.198,E2 15501.198} C_VEL
LIN {X 0,Y 398.331,Z 559.867,A -85,B 0,C 180,E1 15499.122,E2 15499.122} C_VEL
LIN {X 0,Y 394.422,Z 553.93,A -85,B 0,C 180,E1 15496.798,E2 15496.798} C_VEL
LIN {X 0,Y 390.991,Z 548.703,A -85,B 0,C 180,E1 15494.363,E2 15494.363} C_VEL
LIN {X 0,Y 388.14,Z 544.572,A -85,B 0,C 180,E1 15491.893,E2 15491.893} C_VEL
LIN {X 0,Y 385.335,Z 540.036,A -85,B 0,C 180,E1 15488.506,E2 15488.506} C_VEL
LIN {X 0,Y 383.147,Z 536.746,A -85,B 0,C 180,E1 15482.692,E2 15482.692} C_VEL
LIN {X 0,Y 383.454,Z 536.577,A -85,B 0,C 180,E1 15479.402,E2 15479.402} C_VEL
LIN {X 0,Y 384.719,Z 538.082,A -85,B 0,C 180,E1 15476.275,E2 15476.275} C_VEL
LIN {X 0,Y 388.38,Z 541.981,A -85,B 0,C 180,E1 15471.785,E2 15471.785} C_VEL
LIN {X 0,Y 392.814,Z 547.674,A -85,B 0,C 180,E1 15468.176,E2 15468.176} C_VEL
LIN {X 0,Y 397.051,Z 553.267,A -85,B 0,C 180,E1 15465.489,E2 15465.489} C_VEL
LIN {X 0,Y 401.856,Z 559.859,A -85,B 0,C 180,E1 15462.926,E2 15462.926} C_VEL
LIN {X 0,Y 408.571,Z 569.39,A -85,B 0,C 180,E1 15459.889,E2 15459.889} C_VEL
LIN {X 0,Y 416.771,Z 582.034,A -85,B 0,C 180,E1 15456.718,E2 15456.718} C_VEL
LIN {X 0,Y 424.431,Z 594.686,A -85,B 0,C 180,E1 15454.124,E2 15454.124} C_VEL
LIN {X 0,Y 430.922,Z 606.398,A -85,B 0,C 180,E1 15452.123,E2 15452.123} C_VEL
LIN {X 0,Y 414.27,Z 837.139,A -85,B 0,C 180,E1 15448.236,E2 15448.236} C_VEL
LIN {X 0,Y 411.834,Z 859.614,A -85,B 0,C 180,E1 15447.766,E2 15447.766} C_VEL
LIN {X 0,Y 407.778,Z 884.984,A -85,B 0,C 180,E1 15447.049,E2 15447.049} C_VEL
LIN {X 0,Y 403.293,Z 907.039,A -85,B 0,C 180,E1 15446.228,E2 15446.228} C_VEL
LIN {X 0,Y 397.438,Z 930.66,A -85,B 0,C 180,E1 15445.102,E2 15445.102} C_VEL
LIN {X 0,Y 391.625,Z 950.941,A -85,B 0,C 180,E1 15443.909,E2 15443.909} C_VEL
LIN {X 0,Y 384.159,Z 973.592,A -85,B 0,C 180,E1 15442.29,E2 15442.29} C_VEL
LIN {X 0,Y 377.375,Z 992.189,A -85,B 0,C 180,E1 15440.686,E2 15440.686} C_VEL
LIN {X 0,Y 368.863,Z 1013.375,A -85,B 0,C 180,E1 15438.494,E2 15438.494} C_VEL
LIN {X 0,Y 361.4,Z 1030.66,A -85,B 0,C 180,E1 15436.355,E2 15436.355} C_VEL
LIN {X 0,Y 353.025,Z 1048.895,A -85,B 0,C 180,E1 15433.66,E2 15433.66} C_VEL
LIN {X 0,Y 345.806,Z 1064.034,A -85,B 0,C 180,E1 15431.003,E2 15431.003} C_VEL
LIN {X 0,Y 338.194,Z 1079.647,A -85,B 0,C 180,E1 15427.735,E2 15427.735} C_VEL
LIN {X 0,Y 332.155,Z 1091.948,A -85,B 0,C 180,E1 15424.677,E2 15424.677} C_VEL
LIN {X 0,Y 325.694,Z 1105.507,A -85,B 0,C 180,E1 15420.639,E2 15420.639} C_VEL
LIN {X 0,Y 321.172,Z 1115.513,A -85,B 0,C 180,E1 15417.035,E2 15417.035} C_VEL
LIN {X 0,Y 317.079,Z 1125.557,A -85,B 0,C 180,E1 15412.627,E2 15412.627} C_VEL
LIN {X 0,Y 314.706,Z 1132.382,A -85,B 0,C 180,E1 15408.91,E2 15408.91} C_VEL
LIN {X 0,Y 312.985,Z 1138.801,A -85,B 0,C 180,E1 15404.535,E2 15404.535} C_VEL
LIN {X 0,Y 312.204,Z 1143.091,A -85,B 0,C 180,E1 15400.508,E2 15400.508} C_VEL
LIN {X 0,Y 311.98,Z 1145.871,A -85,B 0,C 180,E1 15396.81,E2 15396.81} C_VEL
LIN {X 0,Y 311.956,Z 1147.604,A -85,B 0,C 180,E1 15392.756,E2 15392.756} C_VEL
LIN {X 0,Y 311.976,Z 1147.841,A -85,B 0,C 180,E1 15389.082,E2 15389.082} C_VEL
LIN {X 0,Y 311.96,Z 1147.012,A -85,B 0,C 180,E1 15385.588,E2 15385.588} C_VEL
LIN {X 0,Y 311.999,Z 1145.096,A -85,B 0,C 180,E1 15382.007,E2 15382.007} C_VEL
LIN {X 0,Y 312.472,Z 1141.256,A -85,B 0,C 180,E1 15377.62,E2 15377.62} C_VEL
LIN {X 0,Y 313.545,Z 1136.352,A -85,B 0,C 180,E1 15373.702,E2 15373.702} C_VEL
LIN {X 0,Y 315.667,Z 1129.509,A -85,B 0,C 180,E1 15369.415,E2 15369.415} C_VEL
LIN {X 0,Y 318.773,Z 1121.136,A -85,B 0,C 180,E1 15365.343,E2 15365.343} C_VEL
LIN {X 0,Y 323.078,Z 1111.204,A -85,B 0,C 180,E1 15361.333,E2 15361.333} C_VEL
LIN {X 0,Y 328.507,Z 1099.41,A -85,B 0,C 180,E1 15357.471,E2 15357.471} C_VEL
LIN {X 0,Y 334.731,Z 1086.654,A -85,B 0,C 180,E1 15353.951,E2 15353.951} C_VEL
LIN {X 0,Y 341.867,Z 1071.936,A -85,B 0,C 180,E1 15350.604,E2 15350.604} C_VEL
LIN {X 0,Y 349.626,Z 1056.032,A -85,B 0,C 180,E1 15347.549,E2 15347.549} C_VEL
LIN {X 0,Y 357.276,Z 1039.539,A -85,B 0,C 180,E1 15344.922,E2 15344.922} C_VEL
LIN {X 0,Y 365.369,Z 1021.493,A -85,B 0,C 180,E1 15342.478,E2 15342.478} C_VEL
LIN {X 0,Y 373.228,Z 1002.421,A -85,B 0,C 180,E1 15340.342,E2 15340.342} C_VEL
LIN {X 0,Y 381.003,Z 982.225,A -85,B 0,C 180,E1 15338.429,E2 15338.429} C_VEL
LIN {X 0,Y 388.287,Z 960.973,A -85,B 0,C 180,E1 15336.787,E2 15336.787} C_VEL
LIN {X 0,Y 394.951,Z 939.353,A -85,B 0,C 180,E1 15335.392,E2 15335.392} C_VEL
LIN {X 0,Y 400.556,Z 917.999,A -85,B 0,C 180,E1 15334.283,E2 15334.283} C_VEL
LIN {X 0,Y 405.365,Z 896.898,A -85,B 0,C 180,E1 15333.388,E2 15333.388} C_VEL
LIN {X 0,Y 409.714,Z 872.995,A -85,B 0,C 180,E1 15332.605,E2 15332.605} C_VEL
LIN {X 0,Y 412.763,Z 850.993,A -85,B 0,C 180,E1 15332.054,E2 15332.054} C_VEL
LIN {X 0,Y 415.582,Z 817.485,A -85,B 0,C 180,E1 15331.435,E2 15331.435} C_VEL
LIN {X 0,Y 430.761,Z 606.056,A -85,B 0,C 180,E1 15327.882,E2 15327.882} C_VEL
LIN {X 0,Y 421.765,Z 590.239,A -85,B 0,C 180,E1 15325.073,E2 15325.073} C_VEL
LIN {X 0,Y 413.496,Z 577.079,A -85,B 0,C 180,E1 15322.162,E2 15322.162} C_VEL
LIN {X 0,Y 406.623,Z 566.755,A -85,B 0,C 180,E1 15319.388,E2 15319.388} C_VEL
LIN {X 0,Y 400.535,Z 558.056,A -85,B 0,C 180,E1 15316.534,E2 15316.534} C_VEL
LIN {X 0,Y 395.385,Z 551.14,A -85,B 0,C 180,E1 15313.677,E2 15313.677} C_VEL
LIN {X 0,Y 391.652,Z 546.253,A -85,B 0,C 180,E1 15311.188,E2 15311.188} C_VEL
LIN {X 0,Y 387.582,Z 541.072,A -85,B 0,C 180,E1 15307.71,E2 15307.71} C_VEL
LIN {X 0,Y 383.763,Z 536.84,A -85,B 0,C 180,E1 15302.389,E2 15302.389} C_VEL
LIN {X 0,Y 382.859,Z 535.994,A -85,B 0,C 180,E1 15298.952,E2 15298.952} C_VEL
LIN {X 0,Y 383.077,Z 537.133,A -85,B 0,C 180,E1 15295.509,E2 15295.509} C_VEL
LIN {X 0,Y 385.598,Z 540.584,A -85,B 0,C 180,E1 15290.598,E2 15290.598} C_VEL
LIN {X 0,Y 389.119,Z 546.114,A -85,B 0,C 180,E1 15286.855,E2 15286.855} C_VEL
LIN {X 0,Y 392.051,Z 550.472,A -85,B 0,C 180,E1 15284.543,E2 15284.543} C_VEL
LIN {X 0,Y 396.595,Z 557.238,A -85,B 0,C 180,E1 15281.63,E2 15281.63} C_VEL
LIN {X 0,Y 401.398,Z 564.754,A -85,B 0,C 180,E1 15279.056,E2 15279.056} C_VEL
LIN {X 0,Y 406.083,Z 572.238,A -85,B 0,C 180,E1 15276.875,E2 15276.875} C_VEL
LIN {X 0,Y 412.346,Z 582.534,A -85,B 0,C 180,E1 15274.313,E2 15274.313} C_VEL
LIN {X 0,Y 418.858,Z 593.881,A -85,B 0,C 180,E1 15271.948,E2 15271.948} C_VEL
LIN {X 0,Y 426.426,Z 608.054,A -85,B 0,C 180,E1 15269.473,E2 15269.473} C_VEL
LIN {X 0,Y 429.192,Z 613.672,A -85,B 0,C 180,E1 15268.623,E2 15268.623} C_VEL
LIN {X 0,Y 413.452,Z 844.807,A -85,B 0,C 180,E1 15264.868,E2 15264.868} C_VEL
LIN {X 0,Y 410.352,Z 870.204,A -85,B 0,C 180,E1 15264.302,E2 15264.302} C_VEL
LIN {X 0,Y 406.668,Z 891.662,A -85,B 0,C 180,E1 15263.65,E2 15263.65} C_VEL
LIN {X 0,Y 401.868,Z 913.765,A -85,B 0,C 180,E1 15262.769,E2 15262.769} C_VEL
LIN {X 0,Y 396.504,Z 934.406,A -85,B 0,C 180,E1 15261.736,E2 15261.736} C_VEL
LIN {X 0,Y 389.886,Z 956.153,A -85,B 0,C 180,E1 15260.383,E2 15260.383} C_VEL
LIN {X 0,Y 383.254,Z 975.311,A -85,B 0,C 180,E1 15258.937,E2 15258.937} C_VEL
LIN {X 0,Y 375.441,Z 995.464,A -85,B 0,C 180,E1 15257.088,E2 15257.088} C_VEL
LIN {X 0,Y 368.038,Z 1012.974,A -85,B 0,C 180,E1 15255.161,E2 15255.161} C_VEL
LIN {X 0,Y 359.923,Z 1030.601,A -85,B 0,C 180,E1 15252.827,E2 15252.827} C_VEL
LIN {X 0,Y 352.679,Z 1045.486,A -85,B 0,C 180,E1 15250.485,E2 15250.485} C_VEL
LIN {X 0,Y 344.666,Z 1061.114,A -85,B 0,C 180,E1 15247.533,E2 15247.533} C_VEL
LIN {X 0,Y 337.557,Z 1074.692,A -85,B 0,C 180,E1 15244.456,E2 15244.456} C_VEL
LIN {X 0,Y 331.047,Z 1086.868,A -85,B 0,C 180,E1 15241.097,E2 15241.097} C_VEL
LIN {X 0,Y 325.327,Z 1097.877,A -85,B 0,C 180,E1 15237.453,E2 15237.453} C_VEL
LIN {X 0,Y 320.456,Z 1107.524,A -85,B 0,C 180,E1 15233.459,E2 15233.459} C_VEL
LIN {X 0,Y 316.804,Z 1115.601,A -85,B 0,C 180,E1 15229.317,E2 15229.317} C_VEL
LIN {X 0,Y 314.411,Z 1121.599,A -85,B 0,C 180,E1 15225.305,E2 15225.305} C_VEL
LIN {X 0,Y 312.924,Z 1126.426,A -85,B 0,C 180,E1 15221.053,E2 15221.053} C_VEL
LIN {X 0,Y 312.24,Z 1129.446,A -85,B 0,C 180,E1 15216.99,E2 15216.99} C_VEL
LIN {X 0,Y 312.022,Z 1131.139,A -85,B 0,C 180,E1 15213.123,E2 15213.123} C_VEL
LIN {X 0,Y 311.995,Z 1131.492,A -85,B 0,C 180,E1 15209.082,E2 15209.082} C_VEL
LIN {X 0,Y 312.058,Z 1130.725,A -85,B 0,C 180,E1 15205.59,E2 15205.59} C_VEL
LIN {X 0,Y 312.418,Z 1128.612,A -85,B 0,C 180,E1 15201.477,E2 15201.477} C_VEL
LIN {X 0,Y 313.365,Z 1124.818,A -85,B 0,C 180,E1 15197.281,E2 15197.281} C_VEL
LIN {X 0,Y 315.235,Z 1119.537,A -85,B 0,C 180,E1 15193.033,E2 15193.033} C_VEL
LIN {X 0,Y 318.214,Z 1112.394,A -85,B 0,C 180,E1 15188.817,E2 15188.817} C_VEL
LIN {X 0,Y 322.476,Z 1103.549,A -85,B 0,C 180,E1 15184.666,E2 15184.666} C_VEL
LIN {X 0,Y 327.254,Z 1094.161,A -85,B 0,C 180,E1 15181.134,E2 15181.134} C_VEL
LIN {X 0,Y 333.399,Z 1082.612,A -85,B 0,C 180,E1 15177.531,E2 15177.531} C_VEL
LIN {X 0,Y 339.924,Z 1070.297,A -85,B 0,C 180,E1 15174.379,E2 15174.379} C_VEL
LIN {X 0,Y 347.808,Z 1055.258,A -85,B 0,C 180,E1 15171.177,E2 15171.177} C_VEL
LIN {X 0,Y 355.199,Z 1040.562,A -85,B 0,C 180,E1 15168.583,E2 15168.583} C_VEL
LIN {X 0,Y 363.795,Z 1022.56,A -85,B 0,C 180,E1 15165.943,E2 15165.943} C_VEL
LIN {X 0,Y 371.241,Z 1005.87,A -85,B 0,C 180,E1 15163.905,E2 15163.905} C_VEL
LIN {X 0,Y 379.381,Z 985.884,A -85,B 0,C 180,E1 15161.879,E2 15161.879} C_VEL
LIN {X 0,Y 386.16,Z 967.623,A -85,B 0,C 180,E1 15160.341,E2 15160.341} C_VEL
LIN {X 0,Y 393.054,Z 946.608,A -85,B 0,C 180,E1 15158.882,E2 15158.882} C_VEL
LIN {X 0,Y 398.545,Z 927.494,A -85,B 0,C 180,E1 15157.787,E2 15157.787} C_VEL
LIN {X 0,Y 404.186,Z 904.334,A -85,B 0,C 180,E1 15156.724,E2 15156.724} C_VEL
LIN {X 0,Y 405.533,Z 898.12,A -85,B 0,C 180,E1 15156.481,E2 15156.481} C_VEL
LIN {X 0,Y 406.454,Z 890.893,A -85,B 0,C 180,E1 15156.1,E2 15156.1} C_VEL
LIN {X 0,Y 406.204,Z 872.853,A -85,B 0,C 180,E1 15154.845,E2 15154.845} C_VEL
LIN {X 0,Y 406.828,Z 865.462,A -85,B 0,C 180,E1 15154.528,E2 15154.528} C_VEL
LIN {X 0,Y 409.522,Z 841.689,A -85,B 0,C 180,E1 15154.035,E2 15154.035} C_VEL
LIN {X 0,Y 425.177,Z 617.589,A -85,B 0,C 180,E1 15150.392,E2 15150.392} C_VEL
LIN {X 0,Y 417.494,Z 602.658,A -85,B 0,C 180,E1 15147.841,E2 15147.841} C_VEL
LIN {X 0,Y 411.133,Z 591.313,A -85,B 0,C 180,E1 15145.498,E2 15145.498} C_VEL
LIN {X 0,Y 405.489,Z 581.613,A -85,B 0,C 180,E1 15143.161,E2 15143.161} C_VEL
LIN {X 0,Y 400.453,Z 573.399,A -85,B 0,C 180,E1 15140.805,E2 15140.805} C_VEL
LIN {X 0,Y 395.76,Z 565.788,A -85,B 0,C 180,E1 15138.258,E2 15138.258} C_VEL
LIN {X 0,Y 392.573,Z 561.056,A -85,B 0,C 180,E1 15136.271,E2 15136.271} C_VEL
LIN {X 0,Y 389.65,Z 556.4,A -85,B 0,C 180,E1 15134.11,E2 15134.11} C_VEL
LIN {X 0,Y 386.871,Z 552.288,A -85,B 0,C 180,E1 15131.63,E2 15131.63} C_VEL
LIN {X 0,Y 384.163,Z 547.818,A -85,B 0,C 180,E1 15128.23,E2 15128.23} C_VEL
LIN {X 0,Y 382.163,Z 544.648,A -85,B 0,C 180,E1 15122.549,E2 15122.549} C_VEL
LIN {X 0,Y 382.518,Z 544.552,A -85,B 0,C 180,E1 15119.251,E2 15119.251} C_VEL
LIN {X 0,Y 383.824,Z 546.18,A -85,B 0,C 180,E1 15116.116,E2 15116.116} C_VEL
LIN {X 0,Y 387.168,Z 549.786,A -85,B 0,C 180,E1 15111.983,E2 15111.983} C_VEL
LIN {X 0,Y 391.414,Z 555.363,A -85,B 0,C 180,E1 15108.432,E2 15108.432} C_VEL
LIN {X 0,Y 395.45,Z 560.802,A -85,B 0,C 180,E1 15105.803,E2 15105.803} C_VEL
LIN {X 0,Y 400.155,Z 567.396,A -85,B 0,C 180,E1 15103.225,E2 15103.225} C_VEL
LIN {X 0,Y 406.518,Z 576.651,A -85,B 0,C 180,E1 15100.27,E2 15100.27} C_VEL
LIN {X 0,Y 414.388,Z 589.036,A -85,B 0,C 180,E1 15097.14,E2 15097.14} C_VEL
LIN {X 0,Y 421.81,Z 601.56,A -85,B 0,C 180,E1 15094.555,E2 15094.555} C_VEL
LIN {X 0,Y 426.695,Z 610.618,A -85,B 0,C 180,E1 15092.988,E2 15092.988} C_VEL
LIN {X 0,Y 409.731,Z 839.186,A -85,B 0,C 180,E1 15089.133,E2 15089.133} C_VEL
LIN {X 0,Y 406.927,Z 863.554,A -85,B 0,C 180,E1 15088.612,E2 15088.612} C_VEL
LIN {X 0,Y 402.822,Z 887.41,A -85,B 0,C 180,E1 15087.908,E2 15087.908} C_VEL
LIN {X 0,Y 398.011,Z 910.164,A -85,B 0,C 180,E1 15087.044,E2 15087.044} C_VEL
LIN {X 0,Y 392.201,Z 932.443,A -85,B 0,C 180,E1 15085.952,E2 15085.952} C_VEL
LIN {X 0,Y 385.646,Z 954.528,A -85,B 0,C 180,E1 15084.63,E2 15084.63} C_VEL
LIN {X 0,Y 378.346,Z 975.592,A -85,B 0,C 180,E1 15083.078,E2 15083.078} C_VEL
LIN {X 0,Y 370.527,Z 996.255,A -85,B 0,C 180,E1 15081.25,E2 15081.25} C_VEL
LIN {X 0,Y 362.485,Z 1015.306,A -85,B 0,C 180,E1 15079.205,E2 15079.205} C_VEL
LIN {X 0,Y 353.978,Z 1034.283,A -85,B 0,C 180,E1 15076.785,E2 15076.785} C_VEL
LIN {X 0,Y 345.821,Z 1051.215,A -85,B 0,C 180,E1 15074.172,E2 15074.172} C_VEL
LIN {X 0,Y 337.558,Z 1067.882,A -85,B 0,C 180,E1 15071.117,E2 15071.117} C_VEL
LIN {X 0,Y 330.557,Z 1081.548,A -85,B 0,C 180,E1 15068.103,E2 15068.103} C_VEL
LIN {X 0,Y 323.772,Z 1094.945,A -85,B 0,C 180,E1 15064.628,E2 15064.628} C_VEL
LIN {X 0,Y 317.664,Z 1107.132,A -85,B 0,C 180,E1 15060.761,E2 15060.761} C_VEL
LIN {X 0,Y 312.601,Z 1118.049,A -85,B 0,C 180,E1 15056.603,E2 15056.603} C_VEL
LIN {X 0,Y 308.895,Z 1126.793,A -85,B 0,C 180,E1 15052.456,E2 15052.456} C_VEL
LIN {X 0,Y 306.277,Z 1134.323,A -85,B 0,C 180,E1 15048.068,E2 15048.068} C_VEL
LIN {X 0,Y 304.786,Z 1139.827,A -85,B 0,C 180,E1 15043.815,E2 15043.815} C_VEL
LIN {X 0,Y 304.133,Z 1143.701,A -85,B 0,C 180,E1 15039.844,E2 15039.844} C_VEL
LIN {X 0,Y 303.948,Z 1146.453,A -85,B 0,C 180,E1 15035.474,E2 15035.474} C_VEL
LIN {X 0,Y 303.98,Z 1147.515,A -85,B 0,C 180,E1 15031.885,E2 15031.885} C_VEL
LIN {X 0,Y 303.983,Z 1147.56,A -85,B 0,C 180,E1 15028.492,E2 15028.492} C_VEL
LIN {X 0,Y 303.946,Z 1146.586,A -85,B 0,C 180,E1 15024.904,E2 15024.904} C_VEL
LIN {X 0,Y 304.082,Z 1144.176,A -85,B 0,C 180,E1 15020.728,E2 15020.728} C_VEL
LIN {X 0,Y 304.702,Z 1140.181,A -85,B 0,C 180,E1 15016.527,E2 15016.527} C_VEL
LIN {X 0,Y 306.016,Z 1135.078,A -85,B 0,C 180,E1 15012.506,E2 15012.506} C_VEL
LIN {X 0,Y 308.63,Z 1127.436,A -85,B 0,C 180,E1 15007.908,E2 15007.908} C_VEL
LIN {X 0,Y 311.822,Z 1119.658,A -85,B 0,C 180,E1 15004.145,E2 15004.145} C_VEL
LIN {X 0,Y 317.027,Z 1108.371,A -85,B 0,C 180,E1 14999.693,E2 14999.693} C_VEL
LIN {X 0,Y 322.227,Z 1097.799,A -85,B 0,C 180,E1 14996.258,E2 14996.258} C_VEL
LIN {X 0,Y 329.544,Z 1083.401,A -85,B 0,C 180,E1 14992.365,E2 14992.365} C_VEL
LIN {X 0,Y 336.312,Z 1070.109,A -85,B 0,C 180,E1 14989.374,E2 14989.374} C_VEL
LIN {X 0,Y 345.123,Z 1052.468,A -85,B 0,C 180,E1 14986.062,E2 14986.062} C_VEL
LIN {X 0,Y 352.711,Z 1036.678,A -85,B 0,C 180,E1 14983.588,E2 14983.588} C_VEL
LIN {X 0,Y 361.686,Z 1016.869,A -85,B 0,C 180,E1 14980.999,E2 14980.999} C_VEL
LIN {X 0,Y 369.362,Z 998.705,A -85,B 0,C 180,E1 14979.019,E2 14979.019} C_VEL
LIN {X 0,Y 377.645,Z 977.136,A -85,B 0,C 180,E1 14977.066,E2 14977.066} C_VEL
LIN {X 0,Y 384.684,Z 956.921,A -85,B 0,C 180,E1 14975.554,E2 14975.554} C_VEL
LIN {X 0,Y 391.538,Z 934.287,A -85,B 0,C 180,E1 14974.165,E2 14974.165} C_VEL
LIN {X 0,Y 397.153,Z 912.938,A -85,B 0,C 180,E1 14973.1,E2 14973.1} C_VEL
LIN {X 0,Y 402.445,Z 888.559,A -85,B 0,C 180,E1 14972.147,E2 14972.147} C_VEL
LIN {X 0,Y 406.365,Z 866.049,A -85,B 0,C 180,E1 14971.471,E2 14971.471} C_VEL
LIN {X 0,Y 409.4,Z 841.038,A -85,B 0,C 180,E1 14970.917,E2 14970.917} C_VEL
LIN {X 0,Y 426.273,Z 613.833,A -85,B 0,C 180,E1 14967.079,E2 14967.079} C_VEL
LIN {X 0,Y 426.487,Z 610.152,A -85,B 0,C 180,E1 14967.003,E2 14967.003} C_VEL
LIN {X 0,Y 418.625,Z 596.2,A -85,B 0,C 180,E1 14964.445,E2 14964.445} C_VEL
LIN {X 0,Y 410.919,Z 583.69,A -85,B 0,C 180,E1 14961.632,E2 14961.632} C_VEL
LIN {X 0,Y 404.232,Z 573.412,A -85,B 0,C 180,E1 14958.832,E2 14958.832} C_VEL
LIN {X 0,Y 397.945,Z 564.24,A -85,B 0,C 180,E1 14955.746,E2 14955.746} C_VEL
LIN {X 0,Y 393.698,Z 558.555,A -85,B 0,C 180,E1 14953.288,E2 14953.288} C_VEL
LIN {X 0,Y 390.273,Z 553.95,A -85,B 0,C 180,E1 14950.929,E2 14950.929} C_VEL
LIN {X 0,Y 386.306,Z 548.821,A -85,B 0,C 180,E1 14947.436,E2 14947.436} C_VEL
LIN {X 0,Y 382.723,Z 544.727,A -85,B 0,C 180,E1 14942.246,E2 14942.246} C_VEL
LIN {X 0,Y 381.884,Z 543.935,A -85,B 0,C 180,E1 14938.95,E2 14938.95} C_VEL
LIN {X 0,Y 382.076,Z 545.036,A -85,B 0,C 180,E1 14935.621,E2 14935.621} C_VEL
LIN {X 0,Y 384.514,Z 548.497,A -85,B 0,C 180,E1 14930.722,E2 14930.722} C_VEL
LIN {X 0,Y 387.895,Z 553.948,A -85,B 0,C 180,E1 14927.04,E2 14927.04} C_VEL
LIN {X 0,Y 390.678,Z 558.203,A -85,B 0,C 180,E1 14924.791,E2 14924.791} C_VEL
LIN {X 0,Y 395.017,Z 564.796,A -85,B 0,C 180,E1 14921.936,E2 14921.936} C_VEL
LIN {X 0,Y 399.724,Z 572.361,A -85,B 0,C 180,E1 14919.347,E2 14919.347} C_VEL
LIN {X 0,Y 404.103,Z 579.524,A -85,B 0,C 180,E1 14917.256,E2 14917.256} C_VEL
LIN {X 0,Y 410.075,Z 589.588,A -85,B 0,C 180,E1 14914.741,E2 14914.741} C_VEL
LIN {X 0,Y 416.364,Z 600.806,A -85,B 0,C 180,E1 14912.388,E2 14912.388} C_VEL
LIN {X 0,Y 423.596,Z 614.677,A -85,B 0,C 180,E1 14909.952,E2 14909.952} C_VEL
LIN {X 0,Y 424.991,Z 617.851,A -85,B 0,C 180,E1 14909.496,E2 14909.496} C_VEL
LIN {X 0,Y 409.029,Z 845.421,A -85,B 0,C 180,E1 14905.793,E2 14905.793} C_VEL
LIN {X 0,Y 405.886,Z 870.353,A -85,B 0,C 180,E1 14905.235,E2 14905.235} C_VEL
LIN {X 0,Y 402.087,Z 891.953,A -85,B 0,C 180,E1 14904.58,E2 14904.58} C_VEL
LIN {X 0,Y 397.088,Z 914.331,A -85,B 0,C 180,E1 14903.686,E2 14903.686} C_VEL
LIN {X 0,Y 391.383,Z 935.696,A -85,B 0,C 180,E1 14902.611,E2 14902.611} C_VEL
LIN {X 0,Y 384.595,Z 957.224,A -85,B 0,C 180,E1 14901.257,E2 14901.257} C_VEL
LIN {X 0,Y 377.442,Z 977.293,A -85,B 0,C 180,E1 14899.725,E2 14899.725} C_VEL
LIN {X 0,Y 369.718,Z 996.451,A -85,B 0,C 180,E1 14897.935,E2 14897.935} C_VEL
LIN {X 0,Y 361.6,Z 1015.075,A -85,B 0,C 180,E1 14895.854,E2 14895.854} C_VEL
LIN {X 0,Y 353.432,Z 1032.072,A -85,B 0,C 180,E1 14893.542,E2 14893.542} C_VEL
LIN {X 0,Y 345.178,Z 1048.429,A -85,B 0,C 180,E1 14890.894,E2 14890.894} C_VEL
LIN {X 0,Y 337.425,Z 1062.876,A -85,B 0,C 180,E1 14888.051,E2 14888.051} C_VEL
LIN {X 0,Y 329.769,Z 1076.903,A -85,B 0,C 180,E1 14884.744,E2 14884.744} C_VEL
LIN {X 0,Y 323.271,Z 1088.575,A -85,B 0,C 180,E1 14881.385,E2 14881.385} C_VEL
LIN {X 0,Y 317.091,Z 1099.925,A -85,B 0,C 180,E1 14877.412,E2 14877.412} C_VEL
LIN {X 0,Y 312.678,Z 1108.369,A -85,B 0,C 180,E1 14873.761,E2 14873.761} C_VEL
LIN {X 0,Y 308.739,Z 1116.643,A -85,B 0,C 180,E1 14869.29,E2 14869.29} C_VEL
LIN {X 0,Y 306.41,Z 1122.307,A -85,B 0,C 180,E1 14865.327,E2 14865.327} C_VEL
LIN {X 0,Y 304.855,Z 1127.099,A -85,B 0,C 180,E1 14860.775,E2 14860.775} C_VEL
LIN {X 0,Y 304.244,Z 1129.767,A -85,B 0,C 180,E1 14856.984,E2 14856.984} C_VEL
LIN {X 0,Y 304.02,Z 1131.47,A -85,B 0,C 180,E1 14852.828,E2 14852.828} C_VEL
LIN {X 0,Y 303.999,Z 1131.68,A -85,B 0,C 180,E1 14848.869,E2 14848.869} C_VEL
LIN {X 0,Y 304.075,Z 1130.87,A -85,B 0,C 180,E1 14845.285,E2 14845.285} C_VEL
LIN {X 0,Y 304.472,Z 1128.732,A -85,B 0,C 180,E1 14841.121,E2 14841.121} C_VEL
LIN {X 0,Y 305.472,Z 1125.031,A -85,B 0,C 180,E1 14836.947,E2 14836.947} C_VEL
LIN {X 0,Y 307.466,Z 1119.752,A -85,B 0,C 180,E1 14832.591,E2 14832.591} C_VEL
LIN {X 0,Y 310.623,Z 1112.613,A -85,B 0,C 180,E1 14828.273,E2 14828.273} C_VEL
LIN {X 0,Y 314.893,Z 1104.22,A -85,B 0,C 180,E1 14824.213,E2 14824.213} C_VEL
LIN {X 0,Y 320.125,Z 1094.386,A -85,B 0,C 180,E1 14820.429,E2 14820.429} C_VEL
LIN {X 0,Y 326.725,Z 1082.498,A -85,B 0,C 180,E1 14816.666,E2 14816.666} C_VEL
LIN {X 0,Y 333.628,Z 1070.011,A -85,B 0,C 180,E1 14813.437,E2 14813.437} C_VEL
LIN {X 0,Y 341.904,Z 1054.738,A -85,B 0,C 180,E1 14810.174,E2 14810.174} C_VEL
LIN {X 0,Y 349.641,Z 1039.882,A -85,B 0,C 180,E1 14807.546,E2 14807.546} C_VEL
LIN {X 0,Y 358.279,Z 1022.296,A -85,B 0,C 180,E1 14804.97,E2 14804.97} C_VEL
LIN {X 0,Y 365.96,Z 1005.571,A -85,B 0,C 180,E1 14802.925,E2 14802.925} C_VEL
LIN {X 0,Y 374.056,Z 986.223,A -85,B 0,C 180,E1 14800.961,E2 14800.961} C_VEL
LIN {X 0,Y 381.062,Z 967.851,A -85,B 0,C 180,E1 14799.409,E2 14799.409} C_VEL
LIN {X 0,Y 388.286,Z 946.36,A -85,B 0,C 180,E1 14797.919,E2 14797.919} C_VEL
LIN {X 0,Y 394.261,Z 926.008,A -85,B 0,C 180,E1 14796.764,E2 14796.764} C_VEL
LIN {X 0,Y 399.661,Z 904.096,A -85,B 0,C 180,E1 14795.773,E2 14795.773} C_VEL
LIN {X 0,Y 403.972,Z 882.839,A -85,B 0,C 180,E1 14795.013,E2 14795.013} C_VEL
LIN {X 0,Y 406.828,Z 865.462,A -85,B 0,C 180,E1 14794.528,E2 14794.528} C_VEL
LIN {X 0,Y 407.373,Z 858.013,A -85,B 0,C 180,E1 14794.227,E2 14794.227} C_VEL
LIN {X 0,Y 406.017,Z 838.366,A -85,B 0,C 180,E1 14793.102,E2 14793.102} C_VEL
LIN {X 0,Y 406.102,Z 831.854,A -85,B 0,C 180,E1 14792.905,E2 14792.905} C_VEL
LIN {X 0,Y 421.08,Z 621.638,A -85,B 0,C 180,E1 14789.497,E2 14789.497} C_VEL
LIN {X 0,Y 414.294,Z 608.248,A -85,B 0,C 180,E1 14787.139,E2 14787.139} C_VEL
LIN {X 0,Y 408.458,Z 597.61,A -85,B 0,C 180,E1 14784.901,E2 14784.901} C_VEL
LIN {X 0,Y 402.971,Z 588.04,A -85,B 0,C 180,E1 14782.542,E2 14782.542} C_VEL
LIN {X 0,Y 398.513,Z 580.56,A -85,B 0,C 180,E1 14780.373,E2 14780.373} C_VEL
LIN {X 0,Y 393.948,Z 572.998,A -85,B 0,C 180,E1 14777.809,E2 14777.809} C_VEL
LIN {X 0,Y 390.968,Z 568.463,A -85,B 0,C 180,E1 14775.882,E2 14775.882} C_VEL
LIN {X 0,Y 388.135,Z 563.858,A -85,B 0,C 180,E1 14773.71,E2 14773.71} C_VEL
LIN {X 0,Y 385.611,Z 560.003,A -85,B 0,C 180,E1 14771.366,E2 14771.366} C_VEL
LIN {X 0,Y 383.094,Z 555.701,A -85,B 0,C 180,E1 14768.102,E2 14768.102} C_VEL
LIN {X 0,Y 381.188,Z 552.6,A -85,B 0,C 180,E1 14762.556,E2 14762.556} C_VEL
LIN {X 0,Y 381.543,Z 552.496,A -85,B 0,C 180,E1 14759.249,E2 14759.249} C_VEL
LIN {X 0,Y 382.835,Z 554.149,A -85,B 0,C 180,E1 14756.126,E2 14756.126} C_VEL
LIN {X 0,Y 385.961,Z 557.591,A -85,B 0,C 180,E1 14752.183,E2 14752.183} C_VEL
LIN {X 0,Y 390.025,Z 563.051,A -85,B 0,C 180,E1 14748.69,E2 14748.69} C_VEL
LIN {X 0,Y 393.972,Z 568.516,A -85,B 0,C 180,E1 14746.048,E2 14746.048} C_VEL
LIN {X 0,Y 398.735,Z 575.302,A -85,B 0,C 180,E1 14743.389,E2 14743.389} C_VEL
LIN {X 0,Y 404.707,Z 584.299,A -85,B 0,C 180,E1 14740.554,E2 14740.554} C_VEL
LIN {X 0,Y 412.025,Z 596.052,A -85,B 0,C 180,E1 14737.566,E2 14737.566} C_VEL
LIN {X 0,Y 419.124,Z 608.27,A -85,B 0,C 180,E1 14735.022,E2 14735.022} C_VEL
LIN {X 0,Y 422.552,Z 614.991,A -85,B 0,C 180,E1 14733.868,E2 14733.868} C_VEL
LIN {X 0,Y 405.263,Z 841.621,A -85,B 0,C 180,E1 14730.043,E2 14730.043} C_VEL
LIN {X 0,Y 402.037,Z 867.136,A -85,B 0,C 180,E1 14729.472,E2 14729.472} C_VEL
LIN {X 0,Y 398.096,Z 889.14,A -85,B 0,C 180,E1 14728.812,E2 14728.812} C_VEL
LIN {X 0,Y 392.495,Z 914.088,A -85,B 0,C 180,E1 14727.83,E2 14727.83} C_VEL
LIN {X 0,Y 387.054,Z 934.228,A -85,B 0,C 180,E1 14726.825,E2 14726.825} C_VEL
LIN {X 0,Y 380.027,Z 956.859,A -85,B 0,C 180,E1 14725.441,E2 14725.441} C_VEL
LIN {X 0,Y 373.187,Z 976.041,A -85,B 0,C 180,E1 14724.014,E2 14724.014} C_VEL
LIN {X 0,Y 365.452,Z 995.929,A -85,B 0,C 180,E1 14722.253,E2 14722.253} C_VEL
LIN {X 0,Y 356.918,Z 1015.553,A -85,B 0,C 180,E1 14720.139,E2 14720.139} C_VEL
LIN {X 0,Y 348.381,Z 1034.005,A -85,B 0,C 180,E1 14717.773,E2 14717.773} C_VEL
LIN {X 0,Y 339.934,Z 1050.948,A -85,B 0,C 180,E1 14715.144,E2 14715.144} C_VEL
LIN {X 0,Y 331.354,Z 1067.631,A -85,B 0,C 180,E1 14712.06,E2 14712.06} C_VEL
LIN {X 0,Y 323.881,Z 1081.651,A -85,B 0,C 180,E1 14708.924,E2 14708.924} C_VEL
LIN {X 0,Y 316.646,Z 1095.303,A -85,B 0,C 180,E1 14705.301,E2 14705.301} C_VEL
LIN {X 0,Y 310.432,Z 1107.159,A -85,B 0,C 180,E1 14701.453,E2 14701.453} C_VEL
LIN {X 0,Y 305.215,Z 1117.826,A -85,B 0,C 180,E1 14697.3,E2 14697.3} C_VEL
LIN {X 0,Y 301.278,Z 1126.571,A -85,B 0,C 180,E1 14693.056,E2 14693.056} C_VEL
LIN {X 0,Y 298.475,Z 1134.116,A -85,B 0,C 180,E1 14688.549,E2 14688.549} C_VEL
LIN {X 0,Y 296.883,Z 1139.566,A -85,B 0,C 180,E1 14684.233,E2 14684.233} C_VEL
LIN {X 0,Y 296.159,Z 1143.487,A -85,B 0,C 180,E1 14680.111,E2 14680.111} C_VEL
LIN {X 0,Y 295.954,Z 1146.243,A -85,B 0,C 180,E1 14675.623,E2 14675.623} C_VEL
LIN {X 0,Y 295.981,Z 1147.306,A -85,B 0,C 180,E1 14671.936,E2 14671.936} C_VEL
LIN {X 0,Y 295.986,Z 1147.35,A -85,B 0,C 180,E1 14668.451,E2 14668.451} C_VEL
LIN {X 0,Y 295.948,Z 1146.447,A -85,B 0,C 180,E1 14664.96,E2 14664.96} C_VEL
LIN {X 0,Y 296.073,Z 1144.241,A -85,B 0,C 180,E1 14660.867,E2 14660.867} C_VEL
LIN {X 0,Y 296.735,Z 1140.179,A -85,B 0,C 180,E1 14656.357,E2 14656.357} C_VEL
LIN {X 0,Y 298.082,Z 1135.218,A -85,B 0,C 180,E1 14652.299,E2 14652.299} C_VEL
LIN {X 0,Y 300.859,Z 1127.568,A -85,B 0,C 180,E1 14647.507,E2 14647.507} C_VEL
LIN {X 0,Y 304.199,Z 1119.848,A -85,B 0,C 180,E1 14643.657,E2 14643.657} C_VEL
LIN {X 0,Y 309.397,Z 1109.148,A -85,B 0,C 180,E1 14639.277,E2 14639.277} C_VEL
LIN {X 0,Y 315.041,Z 1098.148,A -85,B 0,C 180,E1 14635.601,E2 14635.601} C_VEL
LIN {X 0,Y 322.179,Z 1084.76,A -85,B 0,C 180,E1 14631.859,E2 14631.859} C_VEL
LIN {X 0,Y 329.643,Z 1070.638,A -85,B 0,C 180,E1 14628.605,E2 14628.605} C_VEL
LIN {X 0,Y 338.19,Z 1054.258,A -85,B 0,C 180,E1 14625.442,E2 14625.442} C_VEL
LIN {X 0,Y 346.307,Z 1037.939,A -85,B 0,C 180,E1 14622.83,E2 14622.83} C_VEL
LIN {X 0,Y 355.251,Z 1019.023,A -85,B 0,C 180,E1 14620.292,E2 14620.292} C_VEL
LIN {X 0,Y 363.144,Z 1000.956,A -85,B 0,C 180,E1 14618.281,E2 14618.281} C_VEL
LIN {X 0,Y 371.64,Z 979.818,A -85,B 0,C 180,E1 14616.312,E2 14616.312} C_VEL
LIN {X 0,Y 378.734,Z 960.142,A -85,B 0,C 180,E1 14614.808,E2 14614.808} C_VEL
LIN {X 0,Y 385.739,Z 938.338,A -85,B 0,C 180,E1 14613.418,E2 14613.418} C_VEL
LIN {X 0,Y 391.626,Z 916.856,A -85,B 0,C 180,E1 14612.317,E2 14612.317} C_VEL
LIN {X 0,Y 397.051,Z 893.767,A -85,B 0,C 180,E1 14611.365,E2 14611.365} C_VEL
LIN {X 0,Y 401.264,Z 870.857,A -85,B 0,C 180,E1 14610.648,E2 14610.648} C_VEL
LIN {X 0,Y 404.617,Z 846.721,A -85,B 0,C 180,E1 14610.068,E2 14610.068} C_VEL
LIN {X 0,Y 409.348,Z 786.649,A -85,B 0,C 180,E1 14609.022,E2 14609.022} C_VEL
LIN {X 0,Y 422.367,Z 614.466,A -85,B 0,C 180,E1 14606.125,E2 14606.125} C_VEL
LIN {X 0,Y 415.357,Z 601.841,A -85,B 0,C 180,E1 14603.742,E2 14603.742} C_VEL
LIN {X 0,Y 408.132,Z 589.903,A -85,B 0,C 180,E1 14600.996,E2 14600.996} C_VEL
LIN {X 0,Y 401.52,Z 579.48,A -85,B 0,C 180,E1 14598.099,E2 14598.099} C_VEL
LIN {X 0,Y 395.655,Z 570.986,A -85,B 0,C 180,E1 14595.088,E2 14595.088} C_VEL
LIN {X 0,Y 392.253,Z 566.234,A -85,B 0,C 180,E1 14593.038,E2 14593.038} C_VEL
LIN {X 0,Y 388.902,Z 561.647,A -85,B 0,C 180,E1 14590.668,E2 14590.668} C_VEL
LIN {X 0,Y 385.182,Z 556.694,A -85,B 0,C 180,E1 14587.308,E2 14587.308} C_VEL
LIN {X 0,Y 381.685,Z 552.614,A -85,B 0,C 180,E1 14582.102,E2 14582.102} C_VEL
LIN {X 0,Y 380.896,Z 551.884,A -85,B 0,C 180,E1 14578.797,E2 14578.797} C_VEL
LIN {X 0,Y 381.134,Z 553.074,A -85,B 0,C 180,E1 14575.486,E2 14575.486} C_VEL
LIN {X 0,Y 383.381,Z 556.307,A -85,B 0,C 180,E1 14570.921,E2 14570.921} C_VEL
LIN {X 0,Y 386.597,Z 561.646,A -85,B 0,C 180,E1 14567.3,E2 14567.3} C_VEL
LIN {X 0,Y 389.218,Z 565.758,A -85,B 0,C 180,E1 14565.114,E2 14565.114} C_VEL
LIN {X 0,Y 393.453,Z 572.354,A -85,B 0,C 180,E1 14562.244,E2 14562.244} C_VEL
LIN {X 0,Y 397.997,Z 579.853,A -85,B 0,C 180,E1 14559.676,E2 14559.676} C_VEL
LIN {X 0,Y 402.141,Z 586.808,A -85,B 0,C 180,E1 14557.64,E2 14557.64} C_VEL
LIN {X 0,Y 407.91,Z 596.793,A -85,B 0,C 180,E1 14555.141,E2 14555.141} C_VEL
LIN {X 0,Y 413.807,Z 607.56,A -85,B 0,C 180,E1 14552.865,E2 14552.865} C_VEL
LIN {X 0,Y 420.701,Z 621.096,A -85,B 0,C 180,E1 14550.47,E2 14550.47} C_VEL
LIN {X 0,Y 420.892,Z 622.069,A -85,B 0,C 180,E1 14550.386,E2 14550.386} C_VEL
LIN {X 0,Y 404.732,Z 845.836,A -85,B 0,C 180,E1 14546.742,E2 14546.742} C_VEL
LIN {X 0,Y 401.529,Z 870.499,A -85,B 0,C 180,E1 14546.189,E2 14546.189} C_VEL
LIN {X 0,Y 397.613,Z 892.243,A -85,B 0,C 180,E1 14545.532,E2 14545.532} C_VEL
LIN {X 0,Y 392.412,Z 914.897,A -85,B 0,C 180,E1 14544.625,E2 14544.625} C_VEL
LIN {X 0,Y 386.823,Z 935.327,A -85,B 0,C 180,E1 14543.601,E2 14543.601} C_VEL
LIN {X 0,Y 380.015,Z 956.514,A -85,B 0,C 180,E1 14542.28,E2 14542.28} C_VEL
LIN {X 0,Y 372.89,Z 976.06,A -85,B 0,C 180,E1 14540.8,E2 14540.8} C_VEL
LIN {X 0,Y 364.649,Z 996.115,A -85,B 0,C 180,E1 14538.944,E2 14538.944} C_VEL
LIN {X 0,Y 356.284,Z 1014.791,A -85,B 0,C 180,E1 14536.859,E2 14536.859} C_VEL
LIN {X 0,Y 347.805,Z 1031.947,A -85,B 0,C 180,E1 14534.523,E2 14534.523} C_VEL
LIN {X 0,Y 339.552,Z 1047.84,A -85,B 0,C 180,E1 14531.948,E2 14531.948} C_VEL
LIN {X 0,Y 331.477,Z 1062.368,A -85,B 0,C 180,E1 14529.083,E2 14529.083} C_VEL
LIN {X 0,Y 323.863,Z 1075.861,A -85,B 0,C 180,E1 14525.917,E2 14525.917} C_VEL
LIN {X 0,Y 316.854,Z 1087.895,A -85,B 0,C 180,E1 14522.444,E2 14522.444} C_VEL
LIN {X 0,Y 310.657,Z 1098.81,A -85,B 0,C 180,E1 14518.658,E2 14518.658} C_VEL
LIN {X 0,Y 305.433,Z 1108.199,A -85,B 0,C 180,E1 14514.567,E2 14514.567} C_VEL
LIN {X 0,Y 301.278,Z 1116.44,A -85,B 0,C 180,E1 14510.077,E2 14510.077} C_VEL
LIN {X 0,Y 298.688,Z 1122.277,A -85,B 0,C 180,E1 14505.933,E2 14505.933} C_VEL
LIN {X 0,Y 296.976,Z 1127.158,A -85,B 0,C 180,E1 14501.261,E2 14501.261} C_VEL
LIN {X 0,Y 296.266,Z 1129.979,A -85,B 0,C 180,E1 14497.174,E2 14497.174} C_VEL
LIN {X 0,Y 296.024,Z 1131.68,A -85,B 0,C 180,E1 14492.904,E2 14492.904} C_VEL
LIN {X 0,Y 296.001,Z 1131.889,A -85,B 0,C 180,E1 14488.839,E2 14488.839} C_VEL
LIN {X 0,Y 296.084,Z 1131.08,A -85,B 0,C 180,E1 14485.157,E2 14485.157} C_VEL
LIN {X 0,Y 296.515,Z 1128.944,A -85,B 0,C 180,E1 14480.881,E2 14480.881} C_VEL
LIN {X 0,Y 297.657,Z 1125.045,A -85,B 0,C 180,E1 14476.4,E2 14476.4} C_VEL
LIN {X 0,Y 299.877,Z 1119.573,A -85,B 0,C 180,E1 14471.858,E2 14471.858} C_VEL
LIN {X 0,Y 303.06,Z 1112.83,A -85,B 0,C 180,E1 14467.702,E2 14467.702} C_VEL
LIN {X 0,Y 307.559,Z 1104.444,A -85,B 0,C 180,E1 14463.551,E2 14463.551} C_VEL
LIN {X 0,Y 313.047,Z 1094.611,A -85,B 0,C 180,E1 14459.691,E2 14459.691} C_VEL
LIN {X 0,Y 319.742,Z 1083.08,A -85,B 0,C 180,E1 14455.96,E2 14455.96} C_VEL
LIN {X 0,Y 326.887,Z 1070.646,A -85,B 0,C 180,E1 14452.683,E2 14452.683} C_VEL
LIN {X 0,Y 335.25,Z 1055.822,A -85,B 0,C 180,E1 14449.444,E2 14449.444} C_VEL
LIN {X 0,Y 343.19,Z 1041.082,A -85,B 0,C 180,E1 14446.789,E2 14446.789} C_VEL
LIN {X 0,Y 352.342,Z 1023.127,A -85,B 0,C 180,E1 14444.112,E2 14444.112} C_VEL
LIN {X 0,Y 360.228,Z 1006.469,A -85,B 0,C 180,E1 14442.054,E2 14442.054} C_VEL
LIN {X 0,Y 368.827,Z 986.56,A -85,B 0,C 180,E1 14440.016,E2 14440.016} C_VEL
LIN {X 0,Y 376.044,Z 968.134,A -85,B 0,C 180,E1 14438.457,E2 14438.457} C_VEL
LIN {X 0,Y 383.403,Z 946.836,A -85,B 0,C 180,E1 14436.977,E2 14436.977} C_VEL
LIN {X 0,Y 389.28,Z 927.339,A -85,B 0,C 180,E1 14435.866,E2 14435.866} C_VEL
LIN {X 0,Y 395.081,Z 904.597,A -85,B 0,C 180,E1 14434.829,E2 14434.829} C_VEL
LIN {X 0,Y 399.461,Z 883.552,A -85,B 0,C 180,E1 14434.076,E2 14434.076} C_VEL
LIN {X 0,Y 403.369,Z 858.989,A -85,B 0,C 180,E1 14433.426,E2 14433.426} C_VEL
LIN {X 0,Y 405.765,Z 836.237,A -85,B 0,C 180,E1 14432.98,E2 14432.98} C_VEL
LIN {X 0,Y 406.102,Z 831.854,A -85,B 0,C 180,E1 14432.905,E2 14432.905} C_VEL
LIN {X 0,Y 406.116,Z 824.281,A -85,B 0,C 180,E1 14432.662,E2 14432.662} C_VEL
LIN {X 0,Y 404.321,Z 804.548,A -85,B 0,C 180,E1 14431.575,E2 14431.575} C_VEL
LIN {X 0,Y 404.416,Z 798.037,A -85,B 0,C 180,E1 14431.377,E2 14431.377} C_VEL
LIN {X 0,Y 417.084,Z 625.617,A -85,B 0,C 180,E1 14428.58,E2 14428.58} C_VEL
LIN {X 0,Y 410.125,Z 611.826,A -85,B 0,C 180,E1 14426.03,E2 14426.03} C_VEL
LIN {X 0,Y 403.413,Z 599.488,A -85,B 0,C 180,E1 14423.248,E2 14423.248} C_VEL
LIN {X 0,Y 397.328,Z 588.886,A -85,B 0,C 180,E1 14420.321,E2 14420.321} C_VEL
LIN {X 0,Y 392.39,Z 580.553,A -85,B 0,C 180,E1 14417.499,E2 14417.499} C_VEL
LIN {X 0,Y 389.381,Z 575.868,A -85,B 0,C 180,E1 14415.49,E2 14415.49} C_VEL
LIN {X 0,Y 386.727,Z 571.434,A -85,B 0,C 180,E1 14413.38,E2 14413.38} C_VEL
LIN {X 0,Y 384.359,Z 567.716,A -85,B 0,C 180,E1 14411.099,E2 14411.099} C_VEL
LIN {X 0,Y 382.027,Z 563.584,A -85,B 0,C 180,E1 14407.974,E2 14407.974} C_VEL
LIN {X 0,Y 380.206,Z 560.503,A -85,B 0,C 180,E1 14402.412,E2 14402.412} C_VEL
LIN {X 0,Y 380.568,Z 560.439,A -85,B 0,C 180,E1 14399.247,E2 14399.247} C_VEL
LIN {X 0,Y 381.784,Z 562.039,A -85,B 0,C 180,E1 14396.246,E2 14396.246} C_VEL
LIN {X 0,Y 384.757,Z 565.395,A -85,B 0,C 180,E1 14392.384,E2 14392.384} C_VEL
LIN {X 0,Y 388.734,Z 570.892,A -85,B 0,C 180,E1 14388.877,E2 14388.877} C_VEL
LIN {X 0,Y 392.39,Z 576.05,A -85,B 0,C 180,E1 14386.367,E2 14386.367} C_VEL
LIN {X 0,Y 397.324,Z 583.199,A -85,B 0,C 180,E1 14383.554,E2 14383.554} C_VEL
LIN {X 0,Y 403.207,Z 592.44,A -85,B 0,C 180,E1 14380.704,E2 14380.704} C_VEL
LIN {X 0,Y 409.77,Z 603.219,A -85,B 0,C 180,E1 14377.965,E2 14377.965} C_VEL
LIN {X 0,Y 416.497,Z 615.036,A -85,B 0,C 180,E1 14375.485,E2 14375.485} C_VEL
LIN {X 0,Y 418.534,Z 619.174,A -85,B 0,C 180,E1 14374.769,E2 14374.769} C_VEL
LIN {X 0,Y 401.007,Z 842.885,A -85,B 0,C 180,E1 14370.995,E2 14370.995} C_VEL
LIN {X 0,Y 397.53,Z 868.973,A -85,B 0,C 180,E1 14370.4,E2 14370.4} C_VEL
LIN {X 0,Y 393.467,Z 890.895,A -85,B 0,C 180,E1 14369.735,E2 14369.735} C_VEL
LIN {X 0,Y 387.744,Z 915.395,A -85,B 0,C 180,E1 14368.758,E2 14368.758} C_VEL
LIN {X 0,Y 382.001,Z 936.014,A -85,B 0,C 180,E1 14367.721,E2 14367.721} C_VEL
LIN {X 0,Y 374.363,Z 959.531,A -85,B 0,C 180,E1 14366.251,E2 14366.251} C_VEL
LIN {X 0,Y 367.193,Z 978.951,A -85,B 0,C 180,E1 14364.778,E2 14364.778} C_VEL
LIN {X 0,Y 358.386,Z 1000.342,A -85,B 0,C 180,E1 14362.801,E2 14362.801} C_VEL
LIN {X 0,Y 350.15,Z 1018.635,A -85,B 0,C 180,E1 14360.768,E2 14360.768} C_VEL
LIN {X 0,Y 341.125,Z 1037.147,A -85,B 0,C 180,E1 14358.289,E2 14358.289} C_VEL
LIN {X 0,Y 333.175,Z 1052.563,A -85,B 0,C 180,E1 14355.829,E2 14355.829} C_VEL
LIN {X 0,Y 323.921,Z 1069.739,A -85,B 0,C 180,E1 14352.533,E2 14352.533} C_VEL
LIN {X 0,Y 316.482,Z 1083.204,A -85,B 0,C 180,E1 14349.423,E2 14349.423} C_VEL
LIN {X 0,Y 308.563,Z 1097.417,A -85,B 0,C 180,E1 14345.454,E2 14345.454} C_VEL
LIN {X 0,Y 302.552,Z 1108.511,A -85,B 0,C 180,E1 14341.7,E2 14341.7} C_VEL
LIN {X 0,Y 297.019,Z 1119.271,A -85,B 0,C 180,E1 14337.248,E2 14337.248} C_VEL
LIN {X 0,Y 293.384,Z 1127.079,A -85,B 0,C 180,E1 14333.287,E2 14333.287} C_VEL
LIN {X 0,Y 290.313,Z 1134.944,A -85,B 0,C 180,E1 14328.266,E2 14328.266} C_VEL
LIN {X 0,Y 288.821,Z 1139.995,A -85,B 0,C 180,E1 14324.025,E2 14324.025} C_VEL
LIN {X 0,Y 288.076,Z 1144.165,A -85,B 0,C 180,E1 14319.187,E2 14319.187} C_VEL
LIN {X 0,Y 287.949,Z 1146.247,A -85,B 0,C 180,E1 14315.18,E2 14315.18} C_VEL
LIN {X 0,Y 287.988,Z 1147.144,A -85,B 0,C 180,E1 14311.592,E2 14311.592} C_VEL
LIN {X 0,Y 287.985,Z 1147.116,A -85,B 0,C 180,E1 14308.209,E2 14308.209} C_VEL
LIN {X 0,Y 287.954,Z 1146.093,A -85,B 0,C 180,E1 14304.42,E2 14304.42} C_VEL
LIN {X 0,Y 288.165,Z 1143.415,A -85,B 0,C 180,E1 14299.807,E2 14299.807} C_VEL
LIN {X 0,Y 288.925,Z 1139.534,A -85,B 0,C 180,E1 14295.571,E2 14295.571} C_VEL
LIN {X 0,Y 290.699,Z 1133.849,A -85,B 0,C 180,E1 14290.927,E2 14290.927} C_VEL
LIN {X 0,Y 293.692,Z 1126.291,A -85,B 0,C 180,E1 14286.313,E2 14286.313} C_VEL
LIN {X 0,Y 297.869,Z 1117.537,A -85,B 0,C 180,E1 14281.969,E2 14281.969} C_VEL
LIN {X 0,Y 303.374,Z 1106.846,A -85,B 0,C 180,E1 14277.728,E2 14277.728} C_VEL
LIN {X 0,Y 310.045,Z 1094.718,A -85,B 0,C 180,E1 14273.731,E2 14273.731} C_VEL
LIN {X 0,Y 317.646,Z 1080.934,A -85,B 0,C 180,E1 14270.047,E2 14270.047} C_VEL
LIN {X 0,Y 325.677,Z 1066.45,A -85,B 0,C 180,E1 14266.791,E2 14266.791} C_VEL
LIN {X 0,Y 334.132,Z 1050.507,A -85,B 0,C 180,E1 14263.847,E2 14263.847} C_VEL
LIN {X 0,Y 343.144,Z 1033.002,A -85,B 0,C 180,E1 14261.127,E2 14261.127} C_VEL
LIN {X 0,Y 351.685,Z 1015.008,A -85,B 0,C 180,E1 14258.828,E2 14258.828} C_VEL
LIN {X 0,Y 360.47,Z 995.31,A -85,B 0,C 180,E1 14256.712,E2 14256.712} C_VEL
LIN {X 0,Y 368.421,Z 975.339,A -85,B 0,C 180,E1 14254.952,E2 14254.952} C_VEL
LIN {X 0,Y 376.231,Z 953.841,A -85,B 0,C 180,E1 14253.376,E2 14253.376} C_VEL
LIN {X 0,Y 382.972,Z 932.136,A -85,B 0,C 180,E1 14252.088,E2 14252.088} C_VEL
LIN {X 0,Y 389.221,Z 909.047,A -85,B 0,C 180,E1 14250.975,E2 14250.975} C_VEL
LIN {X 0,Y 394.255,Z 886.041,A -85,B 0,C 180,E1 14250.118,E2 14250.118} C_VEL
LIN {X 0,Y 398.512,Z 861.643,A -85,B 0,C 180,E1 14249.423,E2 14249.423} C_VEL
LIN {X 0,Y 401.254,Z 838.39,A -85,B 0,C 180,E1 14248.936,E2 14248.936} C_VEL
LIN {X 0,Y 418.368,Z 618.733,A -85,B 0,C 180,E1 14245.234,E2 14245.234} C_VEL
LIN {X 0,Y 411.812,Z 606.851,A -85,B 0,C 180,E1 14242.898,E2 14242.898} C_VEL
LIN {X 0,Y 404.537,Z 594.661,A -85,B 0,C 180,E1 14239.981,E2 14239.981} C_VEL
LIN {X 0,Y 398.301,Z 584.877,A -85,B 0,C 180,E1 14237.081,E2 14237.081} C_VEL
LIN {X 0,Y 393.541,Z 577.874,A -85,B 0,C 180,E1 14234.493,E2 14234.493} C_VEL
LIN {X 0,Y 390.596,Z 573.645,A -85,B 0,C 180,E1 14232.643,E2 14232.643} C_VEL
LIN {X 0,Y 387.538,Z 569.342,A -85,B 0,C 180,E1 14230.405,E2 14230.405} C_VEL
LIN {X 0,Y 384.062,Z 564.568,A -85,B 0,C 180,E1 14227.179,E2 14227.179} C_VEL
LIN {X 0,Y 380.65,Z 560.501,A -85,B 0,C 180,E1 14221.957,E2 14221.957} C_VEL
LIN {X 0,Y 379.921,Z 559.824,A -85,B 0,C 180,E1 14218.794,E2 14218.794} C_VEL
LIN {X 0,Y 380.202,Z 561.123,A -85,B 0,C 180,E1 14215.324,E2 14215.324} C_VEL
LIN {X 0,Y 382.3,Z 564.225,A -85,B 0,C 180,E1 14211.047,E2 14211.047} C_VEL
LIN {X 0,Y 385.384,Z 569.479,A -85,B 0,C 180,E1 14207.488,E2 14207.488} C_VEL
LIN {X 0,Y 387.861,Z 573.485,A -85,B 0,C 180,E1 14205.366,E2 14205.366} C_VEL
LIN {X 0,Y 391.901,Z 579.912,A -85,B 0,C 180,E1 14202.555,E2 14202.555} C_VEL
LIN {X 0,Y 396.545,Z 587.778,A -85,B 0,C 180,E1 14199.868,E2 14199.868} C_VEL
LIN {X 0,Y 400.643,Z 594.859,A -85,B 0,C 180,E1 14197.817,E2 14197.817} C_VEL
LIN {X 0,Y 405.92,Z 604.293,A -85,B 0,C 180,E1 14195.477,E2 14195.477} C_VEL
LIN {X 0,Y 411.806,Z 615.317,A -85,B 0,C 180,E1 14193.152,E2 14193.152} C_VEL
LIN {X 0,Y 416.929,Z 625.747,A -85,B 0,C 180,E1 14191.302,E2 14191.302} C_VEL
LIN {X 0,Y 400.582,Z 845.883,A -85,B 0,C 180,E1 14187.717,E2 14187.717} C_VEL
LIN {X 0,Y 397.286,Z 870.643,A -85,B 0,C 180,E1 14187.164,E2 14187.164} C_VEL
LIN {X 0,Y 393.224,Z 892.683,A -85,B 0,C 180,E1 14186.5,E2 14186.5} C_VEL
LIN {X 0,Y 387.844,Z 915.462,A -85,B 0,C 180,E1 14185.587,E2 14185.587} C_VEL
LIN {X 0,Y 381.88,Z 936.695,A -85,B 0,C 180,E1 14184.519,E2 14184.519} C_VEL
LIN {X 0,Y 374.764,Z 958.037,A -85,B 0,C 180,E1 14183.17,E2 14183.17} C_VEL
LIN {X 0,Y 366.976,Z 978.725,A -85,B 0,C 180,E1 14181.581,E2 14181.581} C_VEL
LIN {X 0,Y 358.817,Z 997.758,A -85,B 0,C 180,E1 14179.777,E2 14179.777} C_VEL
LIN {X 0,Y 350.247,Z 1016.211,A -85,B 0,C 180,E1 14177.68,E2 14177.68} C_VEL
LIN {X 0,Y 341.601,Z 1033.126,A -85,B 0,C 180,E1 14175.339,E2 14175.339} C_VEL
LIN {X 0,Y 332.513,Z 1049.887,A -85,B 0,C 180,E1 14172.546,E2 14172.546} C_VEL
LIN {X 0,Y 324.76,Z 1063.376,A -85,B 0,C 180,E1 14169.822,E2 14169.822} C_VEL
LIN {X 0,Y 316.513,Z 1077.351,A -85,B 0,C 180,E1 14166.435,E2 14166.435} C_VEL
LIN {X 0,Y 309.66,Z 1088.688,A -85,B 0,C 180,E1 14163.073,E2 14163.073} C_VEL
LIN {X 0,Y 302.892,Z 1100.036,A -85,B 0,C 180,E1 14158.978,E2 14158.978} C_VEL
LIN {X 0,Y 297.704,Z 1109.02,A -85,B 0,C 180,E1 14154.927,E2 14154.927} C_VEL
LIN {X 0,Y 293.271,Z 1117.372,A -85,B 0,C 180,E1 14150.142,E2 14150.142} C_VEL
LIN {X 0,Y 290.594,Z 1123.232,A -85,B 0,C 180,E1 14145.773,E2 14145.773} C_VEL
LIN {X 0,Y 288.955,Z 1127.677,A -85,B 0,C 180,E1 14141.174,E2 14141.174} C_VEL
LIN {X 0,Y 288.27,Z 1130.299,A -85,B 0,C 180,E1 14137.173,E2 14137.173} C_VEL
LIN {X 0,Y 288.019,Z 1131.935,A -85,B 0,C 180,E1 14132.587,E2 14132.587} C_VEL
LIN {X 0,Y 288.006,Z 1132.077,A -85,B 0,C 180,E1 14128.607,E2 14128.607} C_VEL
LIN {X 0,Y 288.104,Z 1131.225,A -85,B 0,C 180,E1 14124.823,E2 14124.823} C_VEL
LIN {X 0,Y 288.642,Z 1128.849,A -85,B 0,C 180,E1 14120.227,E2 14120.227} C_VEL
LIN {X 0,Y 289.787,Z 1125.258,A -85,B 0,C 180,E1 14116.023,E2 14116.023} C_VEL
LIN {X 0,Y 292.108,Z 1119.902,A -85,B 0,C 180,E1 14111.437,E2 14111.437} C_VEL
LIN {X 0,Y 295.532,Z 1113.047,A -85,B 0,C 180,E1 14107.102,E2 14107.102} C_VEL
LIN {X 0,Y 300.269,Z 1104.666,A -85,B 0,C 180,E1 14102.857,E2 14102.857} C_VEL
LIN {X 0,Y 306.168,Z 1094.598,A -85,B 0,C 180,E1 14098.832,E2 14098.832} C_VEL
LIN {X 0,Y 313.374,Z 1082.692,A -85,B 0,C 180,E1 14094.947,E2 14094.947} C_VEL
LIN {X 0,Y 320.78,Z 1070.323,A -85,B 0,C 180,E1 14091.662,E2 14091.662} C_VEL
LIN {X 0,Y 329.569,Z 1055.242,A -85,B 0,C 180,E1 14088.361,E2 14088.361} C_VEL
LIN {X 0,Y 337.827,Z 1040.429,A -85,B 0,C 180,E1 14085.692,E2 14085.692} C_VEL
LIN {X 0,Y 347.132,Z 1022.658,A -85,B 0,C 180,E1 14083.052,E2 14083.052} C_VEL
LIN {X 0,Y 355.159,Z 1006.164,A -85,B 0,C 180,E1 14081.017,E2 14081.017} C_VEL
LIN {X 0,Y 364.005,Z 986.17,A -85,B 0,C 180,E1 14078.979,E2 14078.979} C_VEL
LIN {X 0,Y 371.42,Z 967.691,A -85,B 0,C 180,E1 14077.423,E2 14077.423} C_VEL
LIN {X 0,Y 378.821,Z 946.706,A -85,B 0,C 180,E1 14075.974,E2 14075.974} C_VEL
LIN {X 0,Y 384.929,Z 926.896,A -85,B 0,C 180,E1 14074.853,E2 14074.853} C_VEL
LIN {X 0,Y 390.871,Z 903.971,A -85,B 0,C 180,E1 14073.82,E2 14073.82} C_VEL
LIN {X 0,Y 395.36,Z 882.777,A -85,B 0,C 180,E1 14073.071,E2 14073.071} C_VEL
LIN {X 0,Y 399.238,Z 858.655,A -85,B 0,C 180,E1 14072.441,E2 14072.441} C_VEL
LIN {X 0,Y 401.711,Z 835.536,A -85,B 0,C 180,E1 14071.991,E2 14071.991} C_VEL
LIN {X 0,Y 404.416,Z 798.037,A -85,B 0,C 180,E1 14071.377,E2 14071.377} C_VEL
LIN {X 0,Y 404.474,Z 790.466,A -85,B 0,C 180,E1 14071.133,E2 14071.133} C_VEL
LIN {X 0,Y 402.881,Z 770.738,A -85,B 0,C 180,E1 14070.034,E2 14070.034} C_VEL
LIN {X 0,Y 403.008,Z 764.23,A -85,B 0,C 180,E1 14069.834,E2 14069.834} C_VEL
LIN {X 0,Y 413.191,Z 629.805,A -85,B 0,C 180,E1 14067.651,E2 14067.651} C_VEL
LIN {X 0,Y 407.277,Z 617.844,A -85,B 0,C 180,E1 14065.382,E2 14065.382} C_VEL
LIN {X 0,Y 400.971,Z 605.986,A -85,B 0,C 180,E1 14062.661,E2 14062.661} C_VEL
LIN {X 0,Y 395.413,Z 596.052,A -85,B 0,C 180,E1 14059.884,E2 14059.884} C_VEL
LIN {X 0,Y 390.619,Z 587.761,A -85,B 0,C 180,E1 14057.043,E2 14057.043} C_VEL
LIN {X 0,Y 387.812,Z 583.273,A -85,B 0,C 180,E1 14055.094,E2 14055.094} C_VEL
LIN {X 0,Y 385.416,Z 579.13,A -85,B 0,C 180,E1 14053.121,E2 14053.121} C_VEL
LIN {X 0,Y 383.116,Z 575.43,A -85,B 0,C 180,E1 14050.831,E2 14050.831} C_VEL
LIN {X 0,Y 380.874,Z 571.364,A -85,B 0,C 180,E1 14047.694,E2 14047.694} C_VEL
LIN {X 0,Y 379.229,Z 568.372,A -85,B 0,C 180,E1 14042.155,E2 14042.155} C_VEL
LIN {X 0,Y 379.634,Z 568.416,A -85,B 0,C 180,E1 14039.095,E2 14039.095} C_VEL
LIN {X 0,Y 380.977,Z 570.244,A -85,B 0,C 180,E1 14035.936,E2 14035.936} C_VEL
LIN {X 0,Y 383.625,Z 573.321,A -85,B 0,C 180,E1 14032.512,E2 14032.512} C_VEL
LIN {X 0,Y 387.356,Z 578.578,A -85,B 0,C 180,E1 14029.138,E2 14029.138} C_VEL
LIN {X 0,Y 390.93,Z 583.761,A -85,B 0,C 180,E1 14026.616,E2 14026.616} C_VEL
LIN {X 0,Y 395.713,Z 590.852,A -85,B 0,C 180,E1 14023.824,E2 14023.824} C_VEL
LIN {X 0,Y 401.564,Z 600.308,A -85,B 0,C 180,E1 14020.925,E2 14020.925} C_VEL
LIN {X 0,Y 407.622,Z 610.533,A -85,B 0,C 180,E1 14018.335,E2 14018.335} C_VEL
LIN {X 0,Y 414.034,Z 622.044,A -85,B 0,C 180,E1 14015.905,E2 14015.905} C_VEL
LIN {X 0,Y 414.613,Z 623.45,A -85,B 0,C 180,E1 14015.685,E2 14015.685} C_VEL
LIN {X 0,Y 396.97,Z 843.088,A -85,B 0,C 180,E1 14011.988,E2 14011.988} C_VEL
LIN {X 0,Y 393.416,Z 869.117,A -85,B 0,C 180,E1 14011.397,E2 14011.397} C_VEL
LIN {X 0,Y 389.248,Z 891.13,A -85,B 0,C 180,E1 14010.732,E2 14010.732} C_VEL
LIN {X 0,Y 383.405,Z 915.546,A -85,B 0,C 180,E1 14009.763,E2 14009.763} C_VEL
LIN {X 0,Y 377.5,Z 936.26,A -85,B 0,C 180,E1 14008.725,E2 14008.725} C_VEL
LIN {X 0,Y 370.022,Z 958.781,A -85,B 0,C 180,E1 14007.326,E2 14007.326} C_VEL
LIN {X 0,Y 362.743,Z 978.061,A -85,B 0,C 180,E1 14005.875,E2 14005.875} C_VEL
LIN {X 0,Y 353.511,Z 999.971,A -85,B 0,C 180,E1 14003.865,E2 14003.865} C_VEL
LIN {X 0,Y 345.151,Z 1018.027,A -85,B 0,C 180,E1 14001.862,E2 14001.862} C_VEL
LIN {X 0,Y 335.594,Z 1037.056,A -85,B 0,C 180,E1 13999.313,E2 13999.313} C_VEL
LIN {X 0,Y 327.322,Z 1052.561,A -85,B 0,C 180,E1 13996.822,E2 13996.822} C_VEL
LIN {X 0,Y 317.86,Z 1069.489,A -85,B 0,C 180,E1 13993.544,E2 13993.544} C_VEL
LIN {X 0,Y 310.117,Z 1082.96,A -85,B 0,C 180,E1 13990.397,E2 13990.397} C_VEL
LIN {X 0,Y 301.835,Z 1097.184,A -85,B 0,C 180,E1 13986.369,E2 13986.369} C_VEL
LIN {X 0,Y 295.523,Z 1108.281,A -85,B 0,C 180,E1 13982.546,E2 13982.546} C_VEL
LIN {X 0,Y 289.526,Z 1119.338,A -85,B 0,C 180,E1 13977.858,E2 13977.858} C_VEL
LIN {X 0,Y 285.654,Z 1127.221,A -85,B 0,C 180,E1 13973.737,E2 13973.737} C_VEL
LIN {X 0,Y 282.429,Z 1134.991,A -85,B 0,C 180,E1 13968.58,E2 13968.58} C_VEL
LIN {X 0,Y 280.86,Z 1139.995,A -85,B 0,C 180,E1 13964.22,E2 13964.22} C_VEL
LIN {X 0,Y 280.08,Z 1144.073,A -85,B 0,C 180,E1 13959.245,E2 13959.245} C_VEL
LIN {X 0,Y 279.951,Z 1146.036,A -85,B 0,C 180,E1 13955.328,E2 13955.328} C_VEL
LIN {X 0,Y 279.989,Z 1146.934,A -85,B 0,C 180,E1 13951.637,E2 13951.637} C_VEL
LIN {X 0,Y 279.987,Z 1146.907,A -85,B 0,C 180,E1 13948.158,E2 13948.158} C_VEL
LIN {X 0,Y 279.959,Z 1145.882,A -85,B 0,C 180,E1 13944.261,E2 13944.261} C_VEL
LIN {X 0,Y 280.194,Z 1143.201,A -85,B 0,C 180,E1 13939.514,E2 13939.514} C_VEL
LIN {X 0,Y 281.028,Z 1139.317,A -85,B 0,C 180,E1 13935.157,E2 13935.157} C_VEL
LIN {X 0,Y 282.942,Z 1133.63,A -85,B 0,C 180,E1 13930.383,E2 13930.383} C_VEL
LIN {X 0,Y 286.147,Z 1126.067,A -85,B 0,C 180,E1 13925.649,E2 13925.649} C_VEL
LIN {X 0,Y 290.579,Z 1117.311,A -85,B 0,C 180,E1 13921.2,E2 13921.2} C_VEL
LIN {X 0,Y 296.385,Z 1106.613,A -85,B 0,C 180,E1 13916.871,E2 13916.871} C_VEL
LIN {X 0,Y 303.234,Z 1094.739,A -85,B 0,C 180,E1 13912.884,E2 13912.884} C_VEL
LIN {X 0,Y 310.915,Z 1081.4,A -85,B 0,C 180,E1 13909.244,E2 13909.244} C_VEL
LIN {X 0,Y 319.221,Z 1066.987,A -85,B 0,C 180,E1 13905.943,E2 13905.943} C_VEL
LIN {X 0,Y 327.95,Z 1051.177,A -85,B 0,C 180,E1 13902.967,E2 13902.967} C_VEL
LIN {X 0,Y 336.395,Z 1035.313,A -85,B 0,C 180,E1 13900.454,E2 13900.454} C_VEL
LIN {X 0,Y 345.711,Z 1016.547,A -85,B 0,C 180,E1 13897.987,E2 13897.987} C_VEL
LIN {X 0,Y 353.773,Z 999.065,A -85,B 0,C 180,E1 13896.065,E2 13896.065} C_VEL
LIN {X 0,Y 362.835,Z 977.418,A -85,B 0,C 180,E1 13894.095,E2 13894.095} C_VEL
LIN {X 0,Y 369.996,Z 958.406,A -85,B 0,C 180,E1 13892.668,E2 13892.668} C_VEL
LIN {X 0,Y 377.691,Z 935.047,A -85,B 0,C 180,E1 13891.229,E2 13891.229} C_VEL
LIN {X 0,Y 383.667,Z 913.918,A -85,B 0,C 180,E1 13890.18,E2 13890.18} C_VEL
LIN {X 0,Y 389.5,Z 888.975,A -85,B 0,C 180,E1 13889.212,E2 13889.212} C_VEL
LIN {X 0,Y 393.65,Z 866.659,A -85,B 0,C 180,E1 13888.552,E2 13888.552} C_VEL
LIN {X 0,Y 396.946,Z 841.407,A -85,B 0,C 180,E1 13887.996,E2 13887.996} C_VEL
LIN {X 0,Y 414.431,Z 623.062,A -85,B 0,C 180,E1 13884.319,E2 13884.319} C_VEL
LIN {X 0,Y 408.68,Z 612.574,A -85,B 0,C 180,E1 13882.172,E2 13882.172} C_VEL
LIN {X 0,Y 402.261,Z 601.551,A -85,B 0,C 180,E1 13879.494,E2 13879.494} C_VEL
LIN {X 0,Y 396.262,Z 591.91,A -85,B 0,C 180,E1 13876.605,E2 13876.605} C_VEL
LIN {X 0,Y 391.822,Z 585.24,A -85,B 0,C 180,E1 13874.105,E2 13874.105} C_VEL
LIN {X 0,Y 389.065,Z 581.188,A -85,B 0,C 180,E1 13872.316,E2 13872.316} C_VEL
LIN {X 0,Y 386.183,Z 577.037,A -85,B 0,C 180,E1 13870.141,E2 13870.141} C_VEL
LIN {X 0,Y 382.806,Z 572.315,A -85,B 0,C 180,E1 13866.901,E2 13866.901} C_VEL
LIN {X 0,Y 379.617,Z 568.388,A -85,B 0,C 180,E1 13861.811,E2 13861.811} C_VEL
LIN {X 0,Y 378.947,Z 567.765,A -85,B 0,C 180,E1 13858.79,E2 13858.79} C_VEL
LIN {X 0,Y 379.191,Z 569.011,A -85,B 0,C 180,E1 13855.463,E2 13855.463} C_VEL
LIN {X 0,Y 381.171,Z 572.035,A -85,B 0,C 180,E1 13851.249,E2 13851.249} C_VEL
LIN {X 0,Y 384.179,Z 577.311,A -85,B 0,C 180,E1 13847.677,E2 13847.677} C_VEL
LIN {X 0,Y 386.513,Z 581.209,A -85,B 0,C 180,E1 13845.62,E2 13845.62} C_VEL
LIN {X 0,Y 390.472,Z 587.649,A -85,B 0,C 180,E1 13842.797,E2 13842.797} C_VEL
LIN {X 0,Y 395.762,Z 596.758,A -85,B 0,C 180,E1 13839.711,E2 13839.711} C_VEL
LIN {X 0,Y 402.403,Z 608.731,A -85,B 0,C 180,E1 13836.496,E2 13836.496} C_VEL
LIN {X 0,Y 408.702,Z 620.896,A -85,B 0,C 180,E1 13833.872,E2 13833.872} C_VEL
LIN {X 0,Y 413.033,Z 629.96,A -85,B 0,C 180,E1 13832.226,E2 13832.226} C_VEL
LIN {X 0,Y 396.569,Z 845.722,A -85,B 0,C 180,E1 13828.716,E2 13828.716} C_VEL
LIN {X 0,Y 393.204,Z 870.525,A -85,B 0,C 180,E1 13828.166,E2 13828.166} C_VEL
LIN {X 0,Y 389.051,Z 892.597,A -85,B 0,C 180,E1 13827.507,E2 13827.507} C_VEL
LIN {X 0,Y 383.73,Z 914.744,A -85,B 0,C 180,E1 13826.63,E2 13826.63} C_VEL
LIN {X 0,Y 377.766,Z 935.594,A -85,B 0,C 180,E1 13825.594,E2 13825.594} C_VEL
LIN {X 0,Y 370.665,Z 956.658,A -85,B 0,C 180,E1 13824.289,E2 13824.289} C_VEL
LIN {X 0,Y 363.198,Z 976.163,A -85,B 0,C 180,E1 13822.819,E2 13822.819} C_VEL
LIN {X 0,Y 354.569,Z 996.101,A -85,B 0,C 180,E1 13820.979,E2 13820.979} C_VEL
LIN {X 0,Y 346.001,Z 1014.2,A -85,B 0,C 180,E1 13818.96,E2 13818.96} C_VEL
LIN {X 0,Y 336.759,Z 1031.902,A -85,B 0,C 180,E1 13816.549,E2 13816.549} C_VEL
LIN {X 0,Y 327.647,Z 1048.361,A -85,B 0,C 180,E1 13813.848,E2 13813.848} C_VEL
LIN {X 0,Y 319.009,Z 1062.866,A -85,B 0,C 180,E1 13810.926,E2 13810.926} C_VEL
LIN {X 0,Y 310.802,Z 1076.339,A -85,B 0,C 180,E1 13807.68,E2 13807.68} C_VEL
LIN {X 0,Y 303.2,Z 1088.36,A -85,B 0,C 180,E1 13804.099,E2 13804.099} C_VEL
LIN {X 0,Y 296.428,Z 1099.258,A -85,B 0,C 180,E1 13800.172,E2 13800.172} C_VEL
LIN {X 0,Y 290.672,Z 1108.643,A -85,B 0,C 180,E1 13795.905,E2 13795.905} C_VEL
LIN {X 0,Y 286.13,Z 1116.708,A -85,B 0,C 180,E1 13791.311,E2 13791.311} C_VEL
LIN {X 0,Y 283.113,Z 1122.709,A -85,B 0,C 180,E1 13786.834,E2 13786.834} C_VEL
LIN {X 0,Y 281.084,Z 1127.738,A -85,B 0,C 180,E1 13781.699,E2 13781.699} C_VEL
LIN {X 0,Y 280.317,Z 1130.402,A -85,B 0,C 180,E1 13777.584,E2 13777.584} C_VEL
LIN {X 0,Y 280.033,Z 1132.1,A -85,B 0,C 180,E1 13773.07,E2 13773.07} C_VEL
LIN {X 0,Y 280.007,Z 1132.309,A -85,B 0,C 180,E1 13768.772,E2 13768.772} C_VEL
LIN {X 0,Y 280.108,Z 1131.486,A -85,B 0,C 180,E1 13764.837,E2 13764.837} C_VEL
LIN {X 0,Y 280.658,Z 1129.214,A -85,B 0,C 180,E1 13760.154,E2 13760.154} C_VEL
LIN {X 0,Y 281.931,Z 1125.471,A -85,B 0,C 180,E1 13755.625,E2 13755.625} C_VEL
LIN {X 0,Y 284.408,Z 1120.118,A -85,B 0,C 180,E1 13750.916,E2 13750.916} C_VEL
LIN {X 0,Y 288.14,Z 1113.085,A -85,B 0,C 180,E1 13746.366,E2 13746.366} C_VEL
LIN {X 0,Y 293.281,Z 1104.442,A -85,B 0,C 180,E1 13741.934,E2 13741.934} C_VEL
LIN {X 0,Y 299.377,Z 1094.558,A -85,B 0,C 180,E1 13737.924,E2 13737.924} C_VEL
LIN {X 0,Y 307.325,Z 1081.953,A -85,B 0,C 180,E1 13733.792,E2 13733.792} C_VEL
LIN {X 0,Y 314.856,Z 1069.873,A -85,B 0,C 180,E1 13730.569,E2 13730.569} C_VEL
LIN {X 0,Y 324.017,Z 1054.661,A -85,B 0,C 180,E1 13727.242,E2 13727.242} C_VEL
LIN {X 0,Y 332.597,Z 1039.775,A -85,B 0,C 180,E1 13724.561,E2 13724.561} C_VEL
LIN {X 0,Y 341.835,Z 1022.597,A -85,B 0,C 180,E1 13722.015,E2 13722.015} C_VEL
LIN {X 0,Y 349.989,Z 1006.305,A -85,B 0,C 180,E1 13720.002,E2 13720.002} C_VEL
LIN {X 0,Y 358.994,Z 986.506,A -85,B 0,C 180,E1 13717.979,E2 13717.979} C_VEL
LIN {X 0,Y 366.595,Z 968.053,A -85,B 0,C 180,E1 13716.427,E2 13716.427} C_VEL
LIN {X 0,Y 374.432,Z 946.35,A -85,B 0,C 180,E1 13714.933,E2 13714.933} C_VEL
LIN {X 0,Y 380.819,Z 926.057,A -85,B 0,C 180,E1 13713.797,E2 13713.797} C_VEL
LIN {X 0,Y 386.651,Z 903.902,A -85,B 0,C 180,E1 13712.811,E2 13712.811} C_VEL
LIN {X 0,Y 391.293,Z 882.432,A -85,B 0,C 180,E1 13712.059,E2 13712.059} C_VEL
LIN {X 0,Y 395.206,Z 858.478,A -85,B 0,C 180,E1 13711.44,E2 13711.44} C_VEL
LIN {X 0,Y 397.75,Z 835.147,A -85,B 0,C 180,E1 13710.988,E2 13710.988} C_VEL
LIN {X 0,Y 403.008,Z 764.23,A -85,B 0,C 180,E1 13709.834,E2 13709.834} C_VEL
LIN {X 0,Y 403.109,Z 756.662,A -85,B 0,C 180,E1 13709.586,E2 13709.586} C_VEL
LIN {X 0,Y 401.742,Z 736.944,A -85,B 0,C 180,E1 13708.474,E2 13708.474} C_VEL
LIN {X 0,Y 401.911,Z 730.436,A -85,B 0,C 180,E1 13708.274,E2 13708.274} C_VEL
LIN {X 0,Y 409.41,Z 633.921,A -85,B 0,C 180,E1 13706.704,E2 13706.704} C_VEL
LIN {X 0,Y 403.003,Z 620.906,A -85,B 0,C 180,E1 13704.088,E2 13704.088} C_VEL
LIN {X 0,Y 397.439,Z 610.348,A -85,B 0,C 180,E1 13701.511,E2 13701.511} C_VEL
LIN {X 0,Y 392.952,Z 602.258,A -85,B 0,C 180,E1 13699.124,E2 13699.124} C_VEL
LIN {X 0,Y 388.66,Z 594.611,A -85,B 0,C 180,E1 13696.439,E2 13696.439} C_VEL
LIN {X 0,Y 384.445,Z 587.307,A -85,B 0,C 180,E1 13693.154,E2 13693.154} C_VEL
LIN {X 0,Y 381.882,Z 583.142,A -85,B 0,C 180,E1 13690.561,E2 13690.561} C_VEL
LIN {X 0,Y 379.82,Z 579.248,A -85,B 0,C 180,E1 13687.564,E2 13687.564} C_VEL
LIN {X 0,Y 378.254,Z 576.311,A -85,B 0,C 180,E1 13682.121,E2 13682.121} C_VEL
LIN {X 0,Y 378.659,Z 576.361,A -85,B 0,C 180,E1 13679.092,E2 13679.092} C_VEL
LIN {X 0,Y 379.999,Z 578.233,A -85,B 0,C 180,E1 13675.926,E2 13675.926} C_VEL
LIN {X 0,Y 382.431,Z 581.123,A -85,B 0,C 180,E1 13672.715,E2 13672.715} C_VEL
LIN {X 0,Y 385.986,Z 586.264,A -85,B 0,C 180,E1 13669.402,E2 13669.402} C_VEL
LIN {X 0,Y 389.479,Z 591.471,A -85,B 0,C 180,E1 13666.868,E2 13666.868} C_VEL
LIN {X 0,Y 393.981,Z 598.309,A -85,B 0,C 180,E1 13664.167,E2 13664.167} C_VEL
LIN {X 0,Y 399.781,Z 607.918,A -85,B 0,C 180,E1 13661.215,E2 13661.215} C_VEL
LIN {X 0,Y 405.493,Z 617.842,A -85,B 0,C 180,E1 13658.709,E2 13658.709} C_VEL
LIN {X 0,Y 410.805,Z 627.618,A -85,B 0,C 180,E1 13656.62,E2 13656.62} C_VEL
LIN {X 0,Y 393.075,Z 843.084,A -85,B 0,C 180,E1 13653.004,E2 13653.004} C_VEL
LIN {X 0,Y 389.447,Z 869.131,A -85,B 0,C 180,E1 13652.417,E2 13652.417} C_VEL
LIN {X 0,Y 385.194,Z 891.15,A -85,B 0,C 180,E1 13651.758,E2 13651.758} C_VEL
LIN {X 0,Y 379.327,Z 915.192,A -85,B 0,C 180,E1 13650.813,E2 13650.813} C_VEL
LIN {X 0,Y 373.318,Z 935.853,A -85,B 0,C 180,E1 13649.787,E2 13649.787} C_VEL
LIN {X 0,Y 365.346,Z 959.29,A -85,B 0,C 180,E1 13648.338,E2 13648.338} C_VEL
LIN {X 0,Y 358.016,Z 978.211,A -85,B 0,C 180,E1 13646.915,E2 13646.915} C_VEL
LIN {X 0,Y 348.716,Z 999.699,A -85,B 0,C 180,E1 13644.948,E2 13644.948} C_VEL
LIN {X 0,Y 340.436,Z 1017.106,A -85,B 0,C 180,E1 13643.025,E2 13643.025} C_VEL
LIN {X 0,Y 330.277,Z 1036.781,A -85,B 0,C 180,E1 13640.398,E2 13640.398} C_VEL
LIN {X 0,Y 321.868,Z 1052.031,A -85,B 0,C 180,E1 13637.942,E2 13637.942} C_VEL
LIN {X 0,Y 311.903,Z 1069.239,A -85,B 0,C 180,E1 13634.593,E2 13634.593} C_VEL
LIN {X 0,Y 303.841,Z 1082.715,A -85,B 0,C 180,E1 13631.411,E2 13631.411} C_VEL
LIN {X 0,Y 295.189,Z 1096.951,A -85,B 0,C 180,E1 13627.325,E2 13627.325} C_VEL
LIN {X 0,Y 288.56,Z 1108.051,A -85,B 0,C 180,E1 13623.433,E2 13623.433} C_VEL
LIN {X 0,Y 282.387,Z 1118.823,A -85,B 0,C 180,E1 13618.787,E2 13618.787} C_VEL
LIN {X 0,Y 278.283,Z 1126.646,A -85,B 0,C 180,E1 13614.626,E2 13614.626} C_VEL
LIN {X 0,Y 274.76,Z 1134.51,A -85,B 0,C 180,E1 13609.339,E2 13609.339} C_VEL
LIN {X 0,Y 273.019,Z 1139.565,A -85,B 0,C 180,E1 13604.855,E2 13604.855} C_VEL
LIN {X 0,Y 272.137,Z 1143.622,A -85,B 0,C 180,E1 13599.944,E2 13599.944} C_VEL
LIN {X 0,Y 271.955,Z 1145.826,A -85,B 0,C 180,E1 13595.486,E2 13595.486} C_VEL
LIN {X 0,Y 271.991,Z 1146.724,A -85,B 0,C 180,E1 13591.685,E2 13591.685} C_VEL
LIN {X 0,Y 271.988,Z 1146.697,A -85,B 0,C 180,E1 13588.104,E2 13588.104} C_VEL
LIN {X 0,Y 271.966,Z 1145.671,A -85,B 0,C 180,E1 13584.091,E2 13584.091} C_VEL
LIN {X 0,Y 272.226,Z 1142.987,A -85,B 0,C 180,E1 13579.203,E2 13579.203} C_VEL
LIN {X 0,Y 273.139,Z 1139.1,A -85,B 0,C 180,E1 13574.718,E2 13574.718} C_VEL
LIN {X 0,Y 275.211,Z 1133.411,A -85,B 0,C 180,E1 13569.809,E2 13569.809} C_VEL
LIN {X 0,Y 278.644,Z 1125.844,A -85,B 0,C 180,E1 13564.948,E2 13564.948} C_VEL
LIN {X 0,Y 283.347,Z 1117.086,A -85,B 0,C 180,E1 13560.393,E2 13560.393} C_VEL
LIN {X 0,Y 289.466,Z 1106.379,A -85,B 0,C 180,E1 13555.972,E2 13555.972} C_VEL
LIN {X 0,Y 296.657,Z 1094.502,A -85,B 0,C 180,E1 13551.917,E2 13551.917} C_VEL
LIN {X 0,Y 304.671,Z 1081.153,A -85,B 0,C 180,E1 13548.224,E2 13548.224} C_VEL
LIN {X 0,Y 313.549,Z 1066.365,A -85,B 0,C 180,E1 13544.81,E2 13544.81} C_VEL
